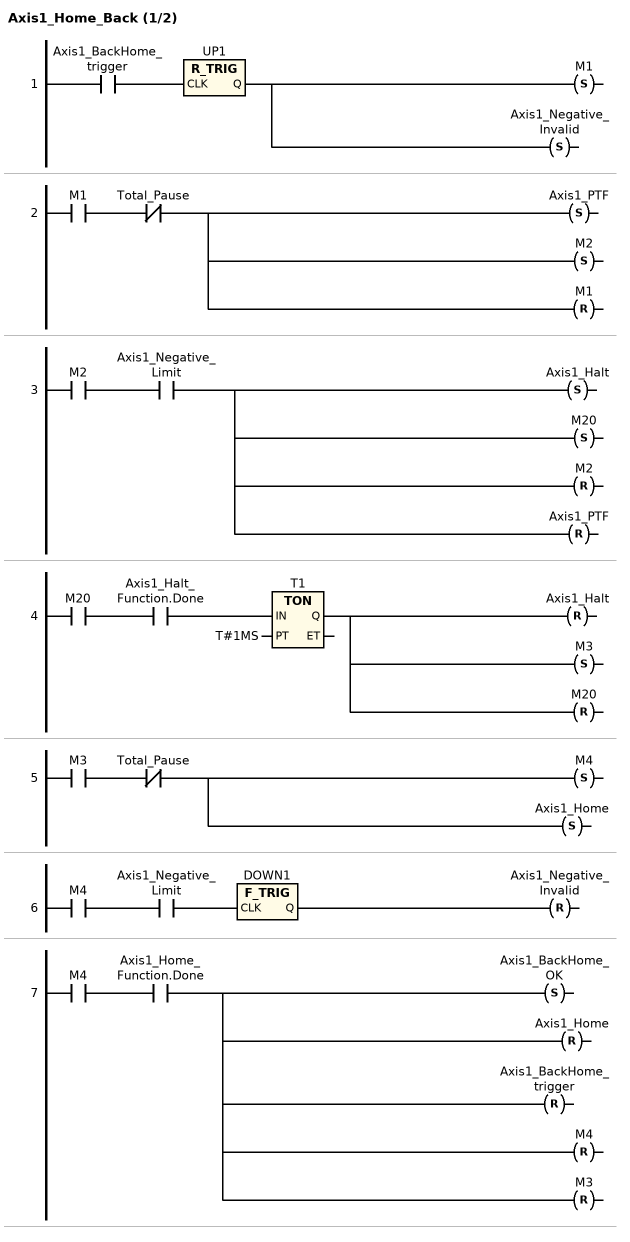
[picture p72: Axis1_Home_Back (LD)]
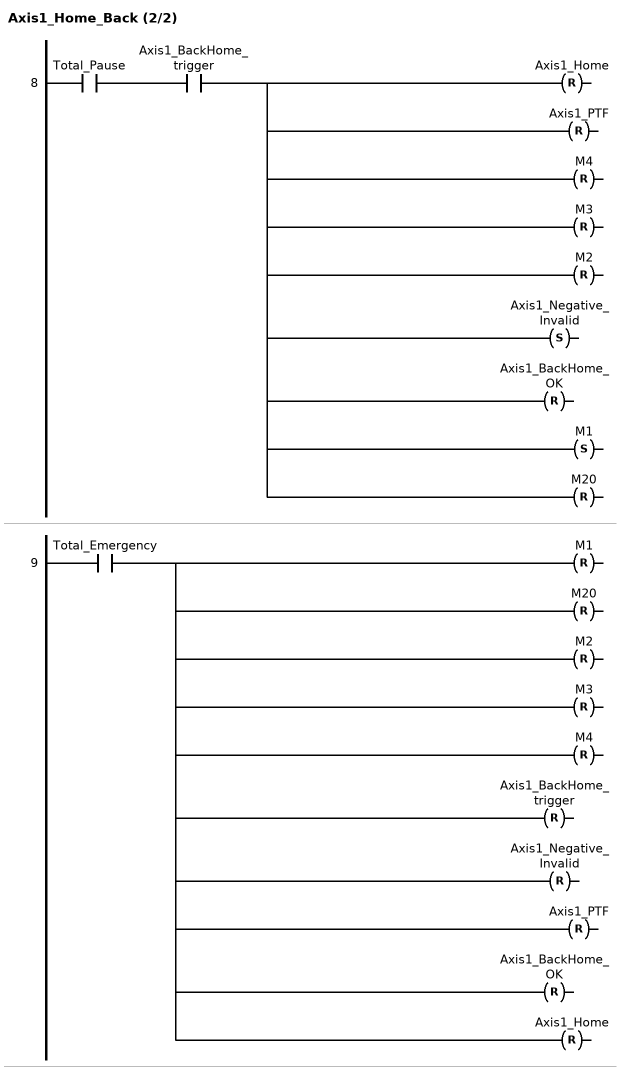
_LD_ (* Ladder Diagram *)
NETWORK 1
	[Axis1_BackHome_trigger] - UP1:R_TRIG(CLK: *) --- (S M1) (S Axis1_Negative_Invalid)
NETWORK 2
	[M1] - [/Total_Pause] --- (S Axis1_PTF) (S M2) (R M1)
NETWORK 3
	[M2] - [Axis1_Negative_Limit] --- (S Axis1_Halt) (S M20) (R M2) (R Axis1_PTF)
NETWORK 4
	[M20] - [Axis1_Halt_Function.Done] - T1:TON(IN: *, PT: T#1MS) --- (R Axis1_Halt) (S M3) (R M20)
NETWORK 5
	[M3] - [/Total_Pause] --- (S M4) (S Axis1_Home)
NETWORK 6
	[M4] - [Axis1_Negative_Limit] - DOWN1:F_TRIG(CLK: *) --- (R Axis1_Negative_Invalid)
NETWORK 7
	[M4] - [Axis1_Home_Function.Done] --- (S Axis1_BackHome_OK) (R Axis1_Home) (R Axis1_BackHome_trigger) (R M4) (R M3)
NETWORK 8
	[Total_Pause] - [Axis1_BackHome_trigger] --- (R Axis1_Home) (R Axis1_PTF) (R M4) (R M3) (R M2) (S Axis1_Negative_Invalid) (R Axis1_BackHome_OK) (S M1) (R M20)
NETWORK 9
	[Total_Emergency] --- (R M1) (R M20) (R M2) (R M3) (R M4) (R Axis1_BackHome_trigger) (R Axis1_Negative_Invalid) (R Axis1_PTF) (R Axis1_BackHome_OK) (R Axis1_Home)
_END_LD_
(* the same logic as Structured Text *)
(* Network 1 *)
UP1(CLK := Axis1_BackHome_trigger);
IF UP1.Q THEN M1 := TRUE; Axis1_Negative_Invalid := TRUE; END_IF;
(* Network 2 *)
_p1 := M1 AND NOT Total_Pause;
IF _p1 THEN Axis1_PTF := TRUE; M2 := TRUE; M1 := FALSE; END_IF;
(* Network 3 *)
_p2 := M2 AND Axis1_Negative_Limit;
IF _p2 THEN Axis1_Halt := TRUE; M20 := TRUE; M2 := FALSE; Axis1_PTF := FALSE; END_IF;
(* Network 4 *)
T1(IN := M20 AND Axis1_Halt_Function.Done, PT := T#1MS);
IF T1.Q THEN Axis1_Halt := FALSE; M3 := TRUE; M20 := FALSE; END_IF;
(* Network 5 *)
IF M3 AND NOT Total_Pause THEN M4 := TRUE; Axis1_Home := TRUE; END_IF;
(* Network 6 *)
DOWN1(CLK := M4 AND Axis1_Negative_Limit);
IF DOWN1.Q THEN Axis1_Negative_Invalid := FALSE; END_IF;
(* Network 7 *)
_p3 := M4 AND Axis1_Home_Function.Done;
IF _p3 THEN Axis1_BackHome_OK := TRUE; Axis1_Home := FALSE; Axis1_BackHome_trigger := FALSE; M4 := FALSE; M3 := FALSE; END_IF;
(* Network 8 *)
IF Total_Pause AND Axis1_BackHome_trigger THEN Axis1_Home := FALSE; Axis1_PTF := FALSE; M4 := FALSE; M3 := FALSE; M2 := FALSE; Axis1_Negative_Invalid := TRUE; Axis1_BackHome_OK := FALSE; M1 := TRUE; M20 := FALSE; END_IF;
(* Network 9 *)
IF Total_Emergency THEN M1 := FALSE; M20 := FALSE; M2 := FALSE; M3 := FALSE; M4 := FALSE; Axis1_BackHome_trigger := FALSE; Axis1_Negative_Invalid := FALSE; Axis1_PTF := FALSE; Axis1_BackHome_OK := FALSE; Axis1_Home := FALSE; END_IF;
END_PROGRAM

(* POU Other_Folder/Home_Back/Axis2_Home_Back, LD *)
PROGRAM Axis2_Home_Back
VAR
	UP1: R_TRIG;
	M1: BOOL;
	M2: BOOL;
	UP2: R_TRIG;
	T1: TON;
	M3: BOOL;
	M4: BOOL;
	DOWN1: F_TRIG;
	M20: BOOL;
END_VAR
VAR (* helpers for the ST form of the networks *)
	_p1 : BOOL;
	_p2 : BOOL;
	_p3 : BOOL;
END_VAR
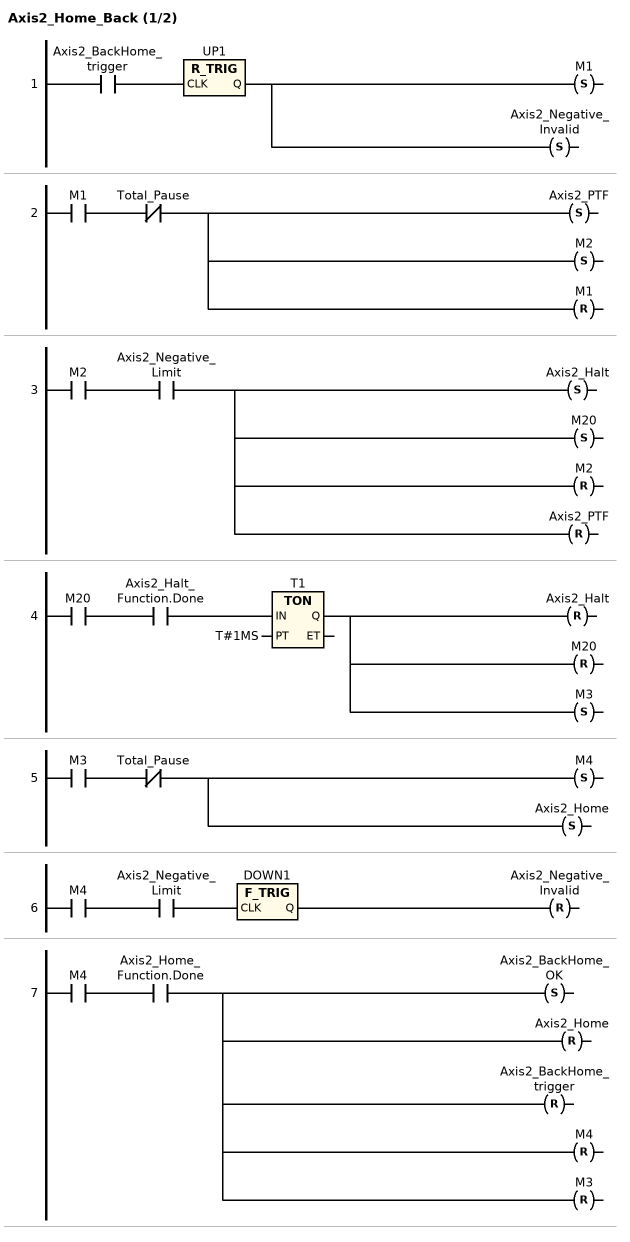
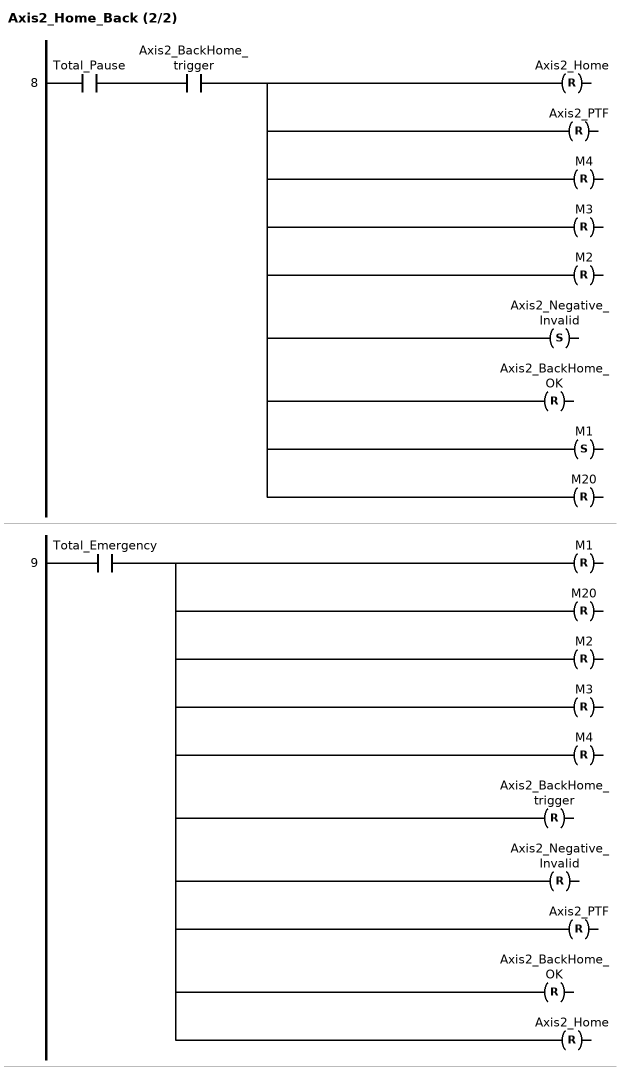
_LD_ (* Ladder Diagram *)
NETWORK 1
	[Axis2_BackHome_trigger] - UP1:R_TRIG(CLK: *) --- (S M1) (S Axis2_Negative_Invalid)
NETWORK 2
	[M1] - [/Total_Pause] --- (S Axis2_PTF) (S M2) (R M1)
NETWORK 3
	[M2] - [Axis2_Negative_Limit] --- (S Axis2_Halt) (S M20) (R M2) (R Axis2_PTF)
NETWORK 4
	[M20] - [Axis2_Halt_Function.Done] - T1:TON(IN: *, PT: T#1MS) --- (R Axis2_Halt) (R M20) (S M3)
NETWORK 5
	[M3] - [/Total_Pause] --- (S M4) (S Axis2_Home)
NETWORK 6
	[M4] - [Axis2_Negative_Limit] - DOWN1:F_TRIG(CLK: *) --- (R Axis2_Negative_Invalid)
NETWORK 7
	[M4] - [Axis2_Home_Function.Done] --- (S Axis2_BackHome_OK) (R Axis2_Home) (R Axis2_BackHome_trigger) (R M4) (R M3)
NETWORK 8
	[Total_Pause] - [Axis2_BackHome_trigger] --- (R Axis2_Home) (R Axis2_PTF) (R M4) (R M3) (R M2) (S Axis2_Negative_Invalid) (R Axis2_BackHome_OK) (S M1) (R M20)
NETWORK 9
	[Total_Emergency] --- (R M1) (R M20) (R M2) (R M3) (R M4) (R Axis2_BackHome_trigger) (R Axis2_Negative_Invalid) (R Axis2_PTF) (R Axis2_BackHome_OK) (R Axis2_Home)
_END_LD_
(* the same logic as Structured Text *)
(* Network 1 *)
UP1(CLK := Axis2_BackHome_trigger);
IF UP1.Q THEN M1 := TRUE; Axis2_Negative_Invalid := TRUE; END_IF;
(* Network 2 *)
_p1 := M1 AND NOT Total_Pause;
IF _p1 THEN Axis2_PTF := TRUE; M2 := TRUE; M1 := FALSE; END_IF;
(* Network 3 *)
_p2 := M2 AND Axis2_Negative_Limit;
IF _p2 THEN Axis2_Halt := TRUE; M20 := TRUE; M2 := FALSE; Axis2_PTF := FALSE; END_IF;
(* Network 4 *)
T1(IN := M20 AND Axis2_Halt_Function.Done, PT := T#1MS);
IF T1.Q THEN Axis2_Halt := FALSE; M20 := FALSE; M3 := TRUE; END_IF;
(* Network 5 *)
IF M3 AND NOT Total_Pause THEN M4 := TRUE; Axis2_Home := TRUE; END_IF;
(* Network 6 *)
DOWN1(CLK := M4 AND Axis2_Negative_Limit);
IF DOWN1.Q THEN Axis2_Negative_Invalid := FALSE; END_IF;
(* Network 7 *)
_p3 := M4 AND Axis2_Home_Function.Done;
IF _p3 THEN Axis2_BackHome_OK := TRUE; Axis2_Home := FALSE; Axis2_BackHome_trigger := FALSE; M4 := FALSE; M3 := FALSE; END_IF;
(* Network 8 *)
IF Total_Pause AND Axis2_BackHome_trigger THEN Axis2_Home := FALSE; Axis2_PTF := FALSE; M4 := FALSE; M3 := FALSE; M2 := FALSE; Axis2_Negative_Invalid := TRUE; Axis2_BackHome_OK := FALSE; M1 := TRUE; M20 := FALSE; END_IF;
(* Network 9 *)
IF Total_Emergency THEN M1 := FALSE; M20 := FALSE; M2 := FALSE; M3 := FALSE; M4 := FALSE; Axis2_BackHome_trigger := FALSE; Axis2_Negative_Invalid := FALSE; Axis2_PTF := FALSE; Axis2_BackHome_OK := FALSE; Axis2_Home := FALSE; END_IF;
END_PROGRAM

(* POU Other_Folder/Home_Back/Axis3_Home_Back, LD *)
PROGRAM Axis3_Home_Back
VAR
	UP1: R_TRIG;
	M1: BOOL;
	M2: BOOL;
	UP2: R_TRIG;
	T1: TON;
	M3: BOOL;
	M4: BOOL;
	DOWN1: F_TRIG;
	M20: BOOL;
END_VAR
VAR (* helpers for the ST form of the networks *)
	_p1 : BOOL;
	_p2 : BOOL;
	_p3 : BOOL;
END_VAR
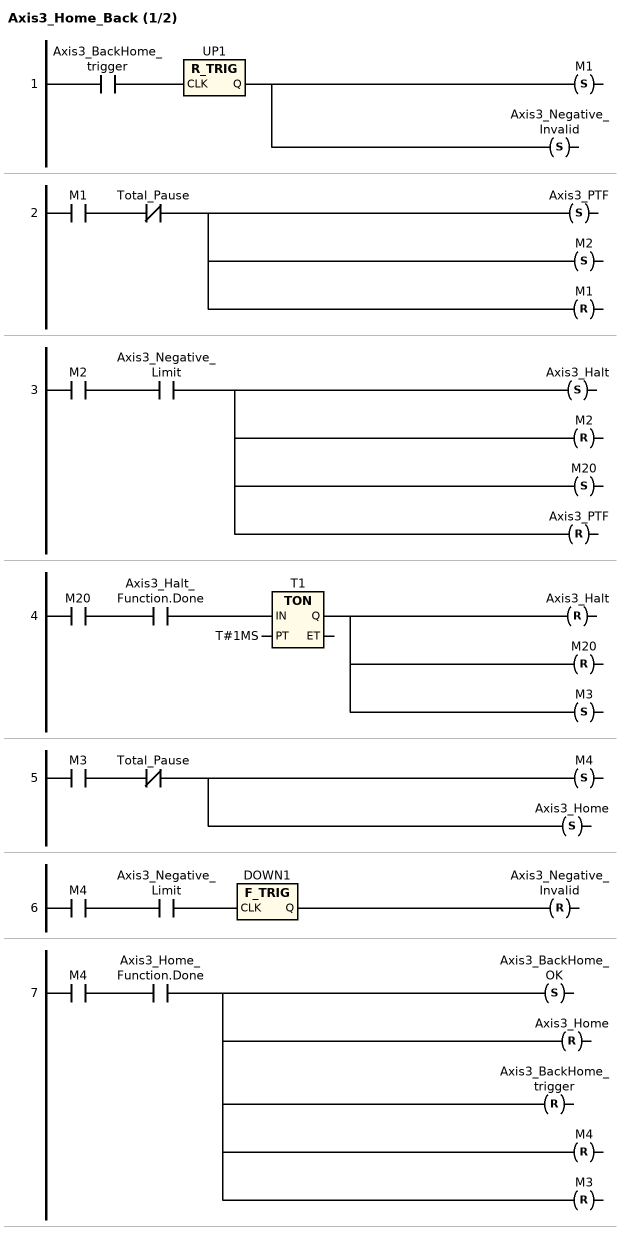
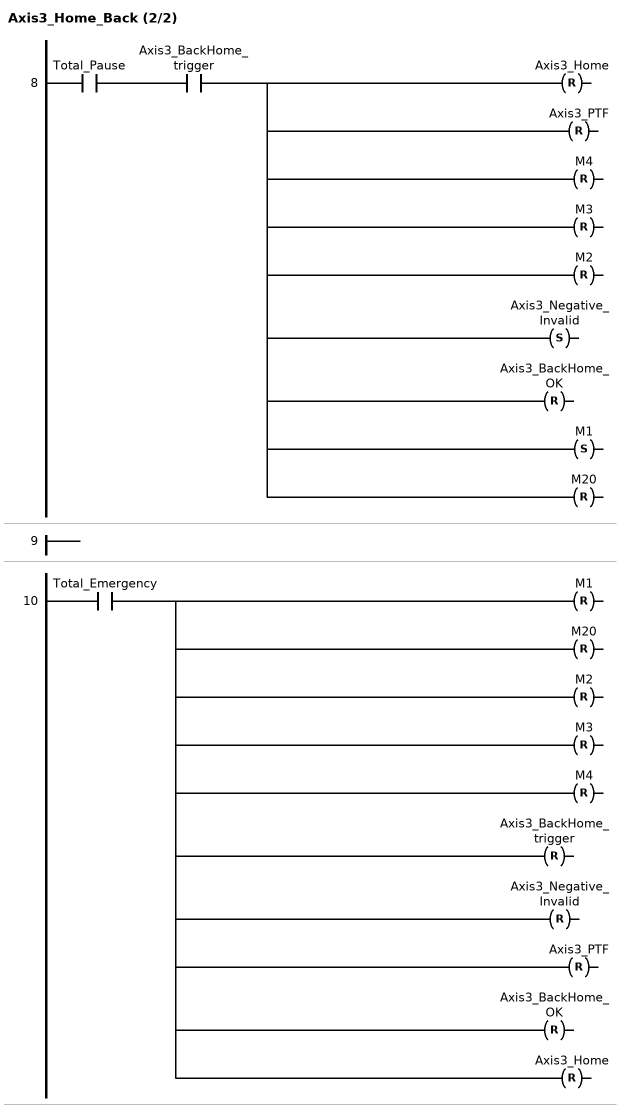
_LD_ (* Ladder Diagram *)
NETWORK 1
	[Axis3_BackHome_trigger] - UP1:R_TRIG(CLK: *) --- (S M1) (S Axis3_Negative_Invalid)
NETWORK 2
	[M1] - [/Total_Pause] --- (S Axis3_PTF) (S M2) (R M1)
NETWORK 3
	[M2] - [Axis3_Negative_Limit] --- (S Axis3_Halt) (R M2) (S M20) (R Axis3_PTF)
NETWORK 4
	[M20] - [Axis3_Halt_Function.Done] - T1:TON(IN: *, PT: T#1MS) --- (R Axis3_Halt) (R M20) (S M3)
NETWORK 5
	[M3] - [/Total_Pause] --- (S M4) (S Axis3_Home)
NETWORK 6
	[M4] - [Axis3_Negative_Limit] - DOWN1:F_TRIG(CLK: *) --- (R Axis3_Negative_Invalid)
NETWORK 7
	[M4] - [Axis3_Home_Function.Done] --- (S Axis3_BackHome_OK) (R Axis3_Home) (R Axis3_BackHome_trigger) (R M4) (R M3)
NETWORK 8
	[Total_Pause] - [Axis3_BackHome_trigger] --- (R Axis3_Home) (R Axis3_PTF) (R M4) (R M3) (R M2) (S Axis3_Negative_Invalid) (R Axis3_BackHome_OK) (S M1) (R M20)
NETWORK 9
	*
NETWORK 10
	[Total_Emergency] --- (R M1) (R M20) (R M2) (R M3) (R M4) (R Axis3_BackHome_trigger) (R Axis3_Negative_Invalid) (R Axis3_PTF) (R Axis3_BackHome_OK) (R Axis3_Home)
_END_LD_
(* the same logic as Structured Text *)
(* Network 1 *)
UP1(CLK := Axis3_BackHome_trigger);
IF UP1.Q THEN M1 := TRUE; Axis3_Negative_Invalid := TRUE; END_IF;
(* Network 2 *)
_p1 := M1 AND NOT Total_Pause;
IF _p1 THEN Axis3_PTF := TRUE; M2 := TRUE; M1 := FALSE; END_IF;
(* Network 3 *)
_p2 := M2 AND Axis3_Negative_Limit;
IF _p2 THEN Axis3_Halt := TRUE; M2 := FALSE; M20 := TRUE; Axis3_PTF := FALSE; END_IF;
(* Network 4 *)
T1(IN := M20 AND Axis3_Halt_Function.Done, PT := T#1MS);
IF T1.Q THEN Axis3_Halt := FALSE; M20 := FALSE; M3 := TRUE; END_IF;
(* Network 5 *)
IF M3 AND NOT Total_Pause THEN M4 := TRUE; Axis3_Home := TRUE; END_IF;
(* Network 6 *)
DOWN1(CLK := M4 AND Axis3_Negative_Limit);
IF DOWN1.Q THEN Axis3_Negative_Invalid := FALSE; END_IF;
(* Network 7 *)
_p3 := M4 AND Axis3_Home_Function.Done;
IF _p3 THEN Axis3_BackHome_OK := TRUE; Axis3_Home := FALSE; Axis3_BackHome_trigger := FALSE; M4 := FALSE; M3 := FALSE; END_IF;
(* Network 8 *)
IF Total_Pause AND Axis3_BackHome_trigger THEN Axis3_Home := FALSE; Axis3_PTF := FALSE; M4 := FALSE; M3 := FALSE; M2 := FALSE; Axis3_Negative_Invalid := TRUE; Axis3_BackHome_OK := FALSE; M1 := TRUE; M20 := FALSE; END_IF;
(* Network 9 *)
(* Network 10 *)
IF Total_Emergency THEN M1 := FALSE; M20 := FALSE; M2 := FALSE; M3 := FALSE; M4 := FALSE; Axis3_BackHome_trigger := FALSE; Axis3_Negative_Invalid := FALSE; Axis3_PTF := FALSE; Axis3_BackHome_OK := FALSE; Axis3_Home := FALSE; END_IF;
END_PROGRAM

(* POU Other_Folder/Home_Back/Axis4_Home_Back, LD *)
PROGRAM Axis4_Home_Back
VAR
	UP1: R_TRIG;
	M1: BOOL;
	M2: BOOL;
	UP2: R_TRIG;
	T1: TON;
	M3: BOOL;
	M4: BOOL;
	DOWN1: F_TRIG;
	M20: BOOL;
END_VAR
VAR (* helpers for the ST form of the networks *)
	_p1 : BOOL;
	_p2 : BOOL;
	_p3 : BOOL;
END_VAR
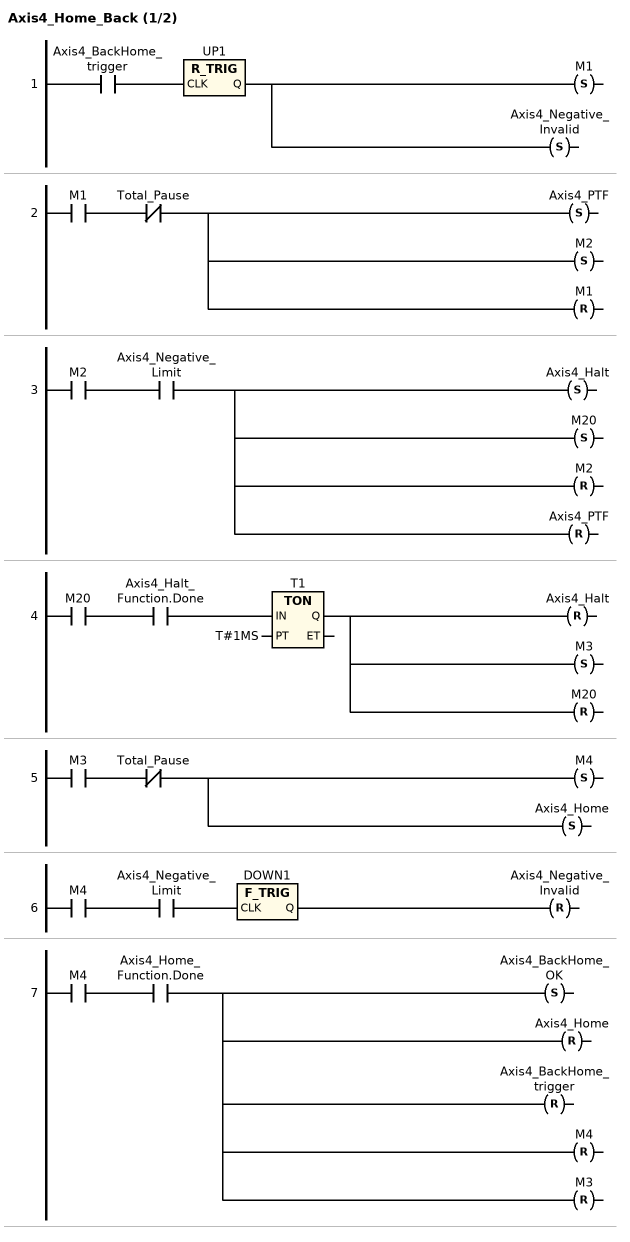
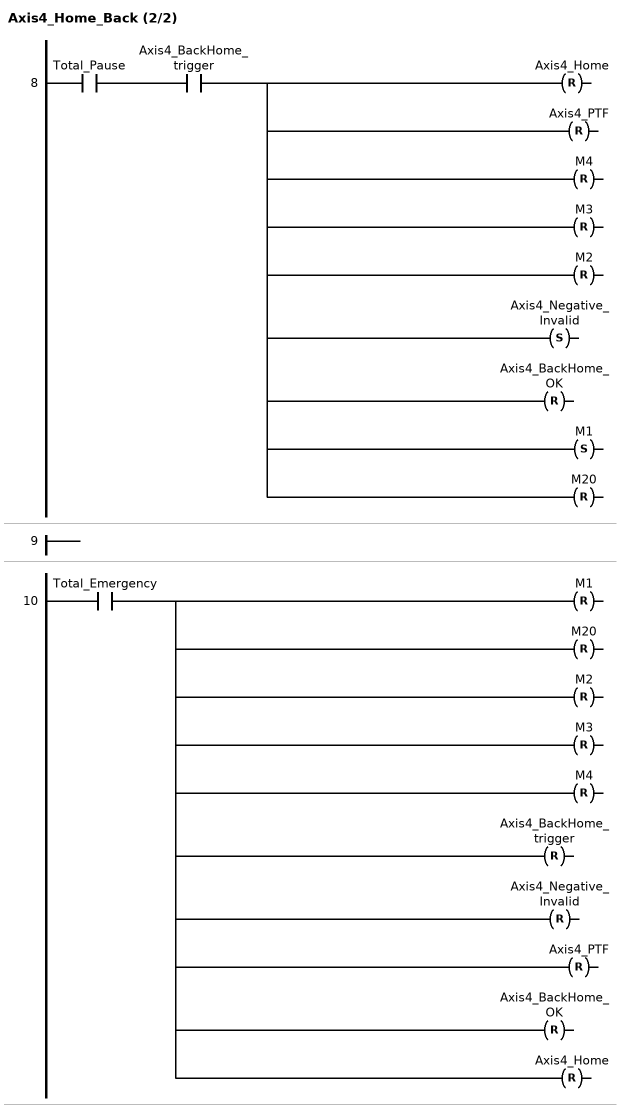
_LD_ (* Ladder Diagram *)
NETWORK 1
	[Axis4_BackHome_trigger] - UP1:R_TRIG(CLK: *) --- (S M1) (S Axis4_Negative_Invalid)
NETWORK 2
	[M1] - [/Total_Pause] --- (S Axis4_PTF) (S M2) (R M1)
NETWORK 3
	[M2] - [Axis4_Negative_Limit] --- (S Axis4_Halt) (S M20) (R M2) (R Axis4_PTF)
NETWORK 4
	[M20] - [Axis4_Halt_Function.Done] - T1:TON(IN: *, PT: T#1MS) --- (R Axis4_Halt) (S M3) (R M20)
NETWORK 5
	[M3] - [/Total_Pause] --- (S M4) (S Axis4_Home)
NETWORK 6
	[M4] - [Axis4_Negative_Limit] - DOWN1:F_TRIG(CLK: *) --- (R Axis4_Negative_Invalid)
NETWORK 7
	[M4] - [Axis4_Home_Function.Done] --- (S Axis4_BackHome_OK) (R Axis4_Home) (R Axis4_BackHome_trigger) (R M4) (R M3)
NETWORK 8
	[Total_Pause] - [Axis4_BackHome_trigger] --- (R Axis4_Home) (R Axis4_PTF) (R M4) (R M3) (R M2) (S Axis4_Negative_Invalid) (R Axis4_BackHome_OK) (S M1) (R M20)
NETWORK 9
	*
NETWORK 10
	[Total_Emergency] --- (R M1) (R M20) (R M2) (R M3) (R M4) (R Axis4_BackHome_trigger) (R Axis4_Negative_Invalid) (R Axis4_PTF) (R Axis4_BackHome_OK) (R Axis4_Home)
_END_LD_
(* the same logic as Structured Text *)
(* Network 1 *)
UP1(CLK := Axis4_BackHome_trigger);
IF UP1.Q THEN M1 := TRUE; Axis4_Negative_Invalid := TRUE; END_IF;
(* Network 2 *)
_p1 := M1 AND NOT Total_Pause;
IF _p1 THEN Axis4_PTF := TRUE; M2 := TRUE; M1 := FALSE; END_IF;
(* Network 3 *)
_p2 := M2 AND Axis4_Negative_Limit;
IF _p2 THEN Axis4_Halt := TRUE; M20 := TRUE; M2 := FALSE; Axis4_PTF := FALSE; END_IF;
(* Network 4 *)
T1(IN := M20 AND Axis4_Halt_Function.Done, PT := T#1MS);
IF T1.Q THEN Axis4_Halt := FALSE; M3 := TRUE; M20 := FALSE; END_IF;
(* Network 5 *)
IF M3 AND NOT Total_Pause THEN M4 := TRUE; Axis4_Home := TRUE; END_IF;
(* Network 6 *)
DOWN1(CLK := M4 AND Axis4_Negative_Limit);
IF DOWN1.Q THEN Axis4_Negative_Invalid := FALSE; END_IF;
(* Network 7 *)
_p3 := M4 AND Axis4_Home_Function.Done;
IF _p3 THEN Axis4_BackHome_OK := TRUE; Axis4_Home := FALSE; Axis4_BackHome_trigger := FALSE; M4 := FALSE; M3 := FALSE; END_IF;
(* Network 8 *)
IF Total_Pause AND Axis4_BackHome_trigger THEN Axis4_Home := FALSE; Axis4_PTF := FALSE; M4 := FALSE; M3 := FALSE; M2 := FALSE; Axis4_Negative_Invalid := TRUE; Axis4_BackHome_OK := FALSE; M1 := TRUE; M20 := FALSE; END_IF;
(* Network 9 *)
(* Network 10 *)
IF Total_Emergency THEN M1 := FALSE; M20 := FALSE; M2 := FALSE; M3 := FALSE; M4 := FALSE; Axis4_BackHome_trigger := FALSE; Axis4_Negative_Invalid := FALSE; Axis4_PTF := FALSE; Axis4_BackHome_OK := FALSE; Axis4_Home := FALSE; END_IF;
END_PROGRAM

(* POU Other_Folder/Home_Back/Axis5_Home_Back, LD *)
PROGRAM Axis5_Home_Back
VAR
	UP1: R_TRIG;
	M1: BOOL;
	M2: BOOL;
	UP2: R_TRIG;
	T1: TON;
	M3: BOOL;
	M4: BOOL;
	DOWN1: F_TRIG;
	M20: BOOL;
END_VAR
VAR (* helpers for the ST form of the networks *)
	_p1 : BOOL;
	_p2 : BOOL;
	_p3 : BOOL;
END_VAR
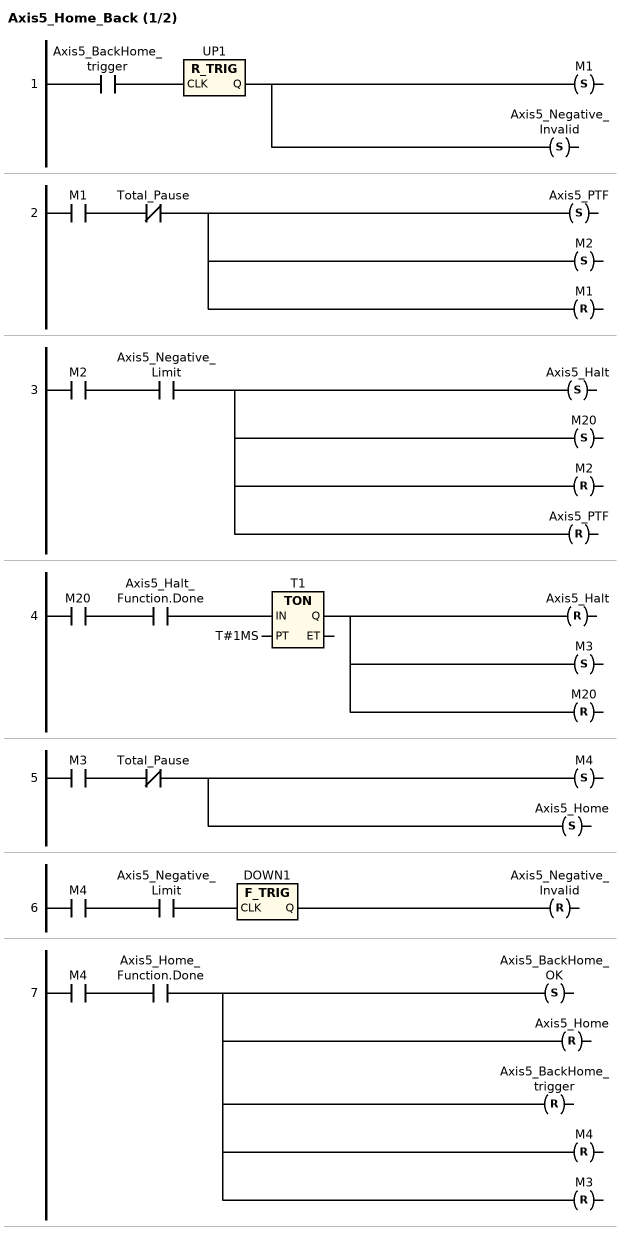
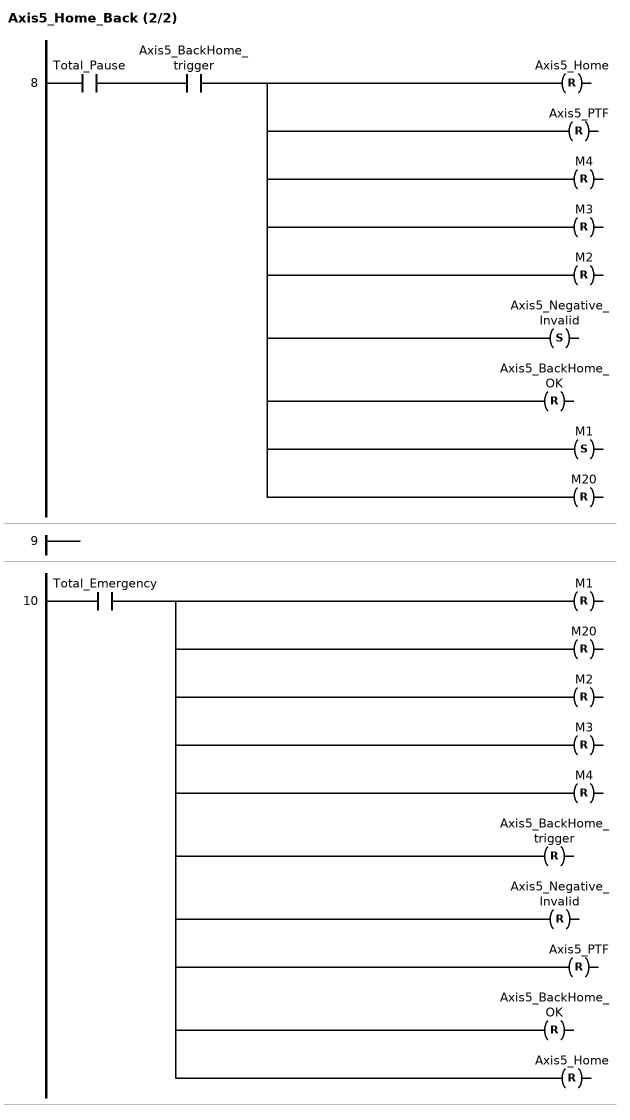
_LD_ (* Ladder Diagram *)
NETWORK 1
	[Axis5_BackHome_trigger] - UP1:R_TRIG(CLK: *) --- (S M1) (S Axis5_Negative_Invalid)
NETWORK 2
	[M1] - [/Total_Pause] --- (S Axis5_PTF) (S M2) (R M1)
NETWORK 3
	[M2] - [Axis5_Negative_Limit] --- (S Axis5_Halt) (S M20) (R M2) (R Axis5_PTF)
NETWORK 4
	[M20] - [Axis5_Halt_Function.Done] - T1:TON(IN: *, PT: T#1MS) --- (R Axis5_Halt) (S M3) (R M20)
NETWORK 5
	[M3] - [/Total_Pause] --- (S M4) (S Axis5_Home)
NETWORK 6
	[M4] - [Axis5_Negative_Limit] - DOWN1:F_TRIG(CLK: *) --- (R Axis5_Negative_Invalid)
NETWORK 7
	[M4] - [Axis5_Home_Function.Done] --- (S Axis5_BackHome_OK) (R Axis5_Home) (R Axis5_BackHome_trigger) (R M4) (R M3)
NETWORK 8
	[Total_Pause] - [Axis5_BackHome_trigger] --- (R Axis5_Home) (R Axis5_PTF) (R M4) (R M3) (R M2) (S Axis5_Negative_Invalid) (R Axis5_BackHome_OK) (S M1) (R M20)
NETWORK 9
	*
NETWORK 10
	[Total_Emergency] --- (R M1) (R M20) (R M2) (R M3) (R M4) (R Axis5_BackHome_trigger) (R Axis5_Negative_Invalid) (R Axis5_PTF) (R Axis5_BackHome_OK) (R Axis5_Home)
_END_LD_
(* the same logic as Structured Text *)
(* Network 1 *)
UP1(CLK := Axis5_BackHome_trigger);
IF UP1.Q THEN M1 := TRUE; Axis5_Negative_Invalid := TRUE; END_IF;
(* Network 2 *)
_p1 := M1 AND NOT Total_Pause;
IF _p1 THEN Axis5_PTF := TRUE; M2 := TRUE; M1 := FALSE; END_IF;
(* Network 3 *)
_p2 := M2 AND Axis5_Negative_Limit;
IF _p2 THEN Axis5_Halt := TRUE; M20 := TRUE; M2 := FALSE; Axis5_PTF := FALSE; END_IF;
(* Network 4 *)
T1(IN := M20 AND Axis5_Halt_Function.Done, PT := T#1MS);
IF T1.Q THEN Axis5_Halt := FALSE; M3 := TRUE; M20 := FALSE; END_IF;
(* Network 5 *)
IF M3 AND NOT Total_Pause THEN M4 := TRUE; Axis5_Home := TRUE; END_IF;
(* Network 6 *)
DOWN1(CLK := M4 AND Axis5_Negative_Limit);
IF DOWN1.Q THEN Axis5_Negative_Invalid := FALSE; END_IF;
(* Network 7 *)
_p3 := M4 AND Axis5_Home_Function.Done;
IF _p3 THEN Axis5_BackHome_OK := TRUE; Axis5_Home := FALSE; Axis5_BackHome_trigger := FALSE; M4 := FALSE; M3 := FALSE; END_IF;
(* Network 8 *)
IF Total_Pause AND Axis5_BackHome_trigger THEN Axis5_Home := FALSE; Axis5_PTF := FALSE; M4 := FALSE; M3 := FALSE; M2 := FALSE; Axis5_Negative_Invalid := TRUE; Axis5_BackHome_OK := FALSE; M1 := TRUE; M20 := FALSE; END_IF;
(* Network 9 *)
(* Network 10 *)
IF Total_Emergency THEN M1 := FALSE; M20 := FALSE; M2 := FALSE; M3 := FALSE; M4 := FALSE; Axis5_BackHome_trigger := FALSE; Axis5_Negative_Invalid := FALSE; Axis5_PTF := FALSE; Axis5_BackHome_OK := FALSE; Axis5_Home := FALSE; END_IF;
END_PROGRAM

(* POU Other_Folder/Home_Back/Axis6_Home_Back, LD *)
PROGRAM Axis6_Home_Back
VAR
	UP1: R_TRIG;
	M1: BOOL;
	M2: BOOL;
	UP2: R_TRIG;
	T1: TON;
	M3: BOOL;
	M4: BOOL;
	DOWN1: F_TRIG;
	M20: BOOL;
END_VAR
VAR (* helpers for the ST form of the networks *)
	_p1 : BOOL;
	_p2 : BOOL;
	_p3 : BOOL;
END_VAR
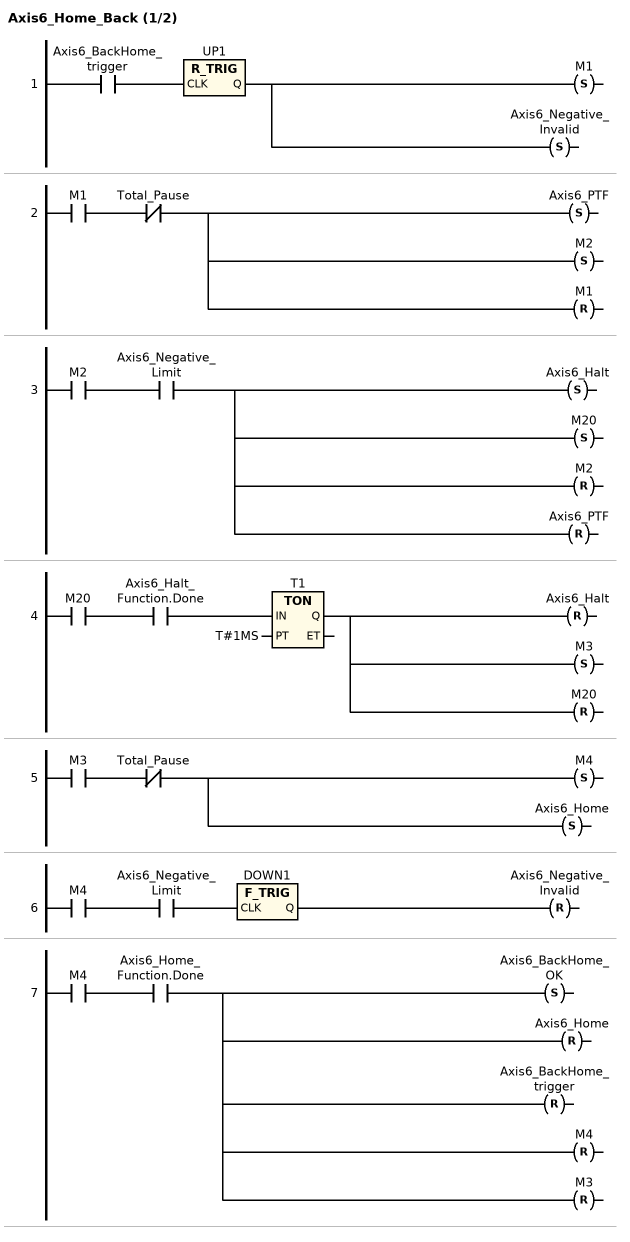
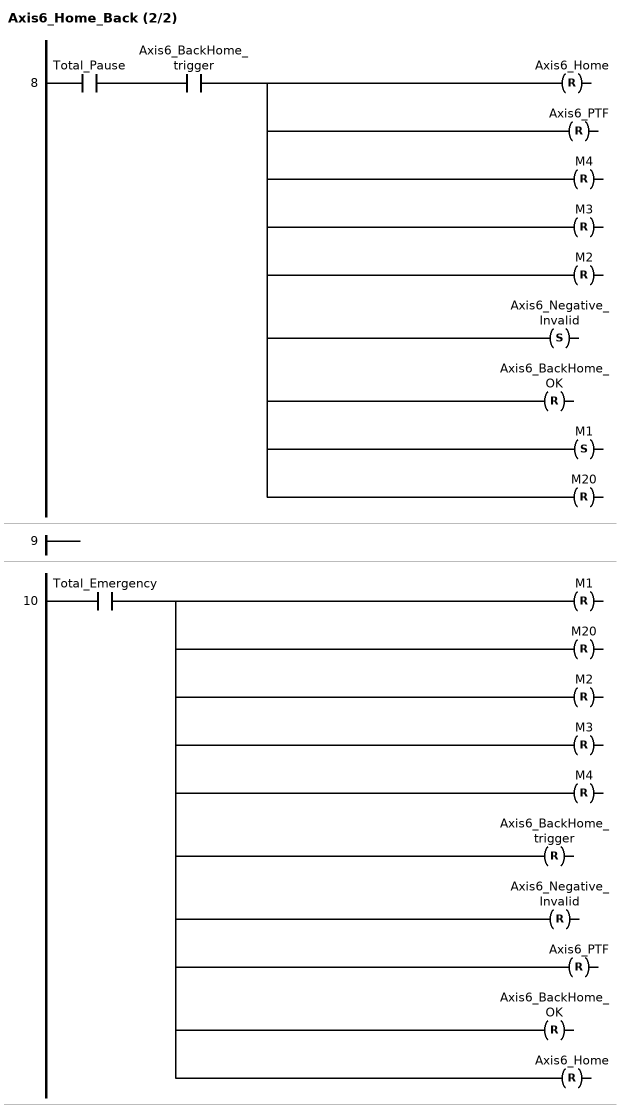
_LD_ (* Ladder Diagram *)
NETWORK 1
	[Axis6_BackHome_trigger] - UP1:R_TRIG(CLK: *) --- (S M1) (S Axis6_Negative_Invalid)
NETWORK 2
	[M1] - [/Total_Pause] --- (S Axis6_PTF) (S M2) (R M1)
NETWORK 3
	[M2] - [Axis6_Negative_Limit] --- (S Axis6_Halt) (S M20) (R M2) (R Axis6_PTF)
NETWORK 4
	[M20] - [Axis6_Halt_Function.Done] - T1:TON(IN: *, PT: T#1MS) --- (R Axis6_Halt) (S M3) (R M20)
NETWORK 5
	[M3] - [/Total_Pause] --- (S M4) (S Axis6_Home)
NETWORK 6
	[M4] - [Axis6_Negative_Limit] - DOWN1:F_TRIG(CLK: *) --- (R Axis6_Negative_Invalid)
NETWORK 7
	[M4] - [Axis6_Home_Function.Done] --- (S Axis6_BackHome_OK) (R Axis6_Home) (R Axis6_BackHome_trigger) (R M4) (R M3)
NETWORK 8
	[Total_Pause] - [Axis6_BackHome_trigger] --- (R Axis6_Home) (R Axis6_PTF) (R M4) (R M3) (R M2) (S Axis6_Negative_Invalid) (R Axis6_BackHome_OK) (S M1) (R M20)
NETWORK 9
	*
NETWORK 10
	[Total_Emergency] --- (R M1) (R M20) (R M2) (R M3) (R M4) (R Axis6_BackHome_trigger) (R Axis6_Negative_Invalid) (R Axis6_PTF) (R Axis6_BackHome_OK) (R Axis6_Home)
_END_LD_
(* the same logic as Structured Text *)
(* Network 1 *)
UP1(CLK := Axis6_BackHome_trigger);
IF UP1.Q THEN M1 := TRUE; Axis6_Negative_Invalid := TRUE; END_IF;
(* Network 2 *)
_p1 := M1 AND NOT Total_Pause;
IF _p1 THEN Axis6_PTF := TRUE; M2 := TRUE; M1 := FALSE; END_IF;
(* Network 3 *)
_p2 := M2 AND Axis6_Negative_Limit;
IF _p2 THEN Axis6_Halt := TRUE; M20 := TRUE; M2 := FALSE; Axis6_PTF := FALSE; END_IF;
(* Network 4 *)
T1(IN := M20 AND Axis6_Halt_Function.Done, PT := T#1MS);
IF T1.Q THEN Axis6_Halt := FALSE; M3 := TRUE; M20 := FALSE; END_IF;
(* Network 5 *)
IF M3 AND NOT Total_Pause THEN M4 := TRUE; Axis6_Home := TRUE; END_IF;
(* Network 6 *)
DOWN1(CLK := M4 AND Axis6_Negative_Limit);
IF DOWN1.Q THEN Axis6_Negative_Invalid := FALSE; END_IF;
(* Network 7 *)
_p3 := M4 AND Axis6_Home_Function.Done;
IF _p3 THEN Axis6_BackHome_OK := TRUE; Axis6_Home := FALSE; Axis6_BackHome_trigger := FALSE; M4 := FALSE; M3 := FALSE; END_IF;
(* Network 8 *)
IF Total_Pause AND Axis6_BackHome_trigger THEN Axis6_Home := FALSE; Axis6_PTF := FALSE; M4 := FALSE; M3 := FALSE; M2 := FALSE; Axis6_Negative_Invalid := TRUE; Axis6_BackHome_OK := FALSE; M1 := TRUE; M20 := FALSE; END_IF;
(* Network 9 *)
(* Network 10 *)
IF Total_Emergency THEN M1 := FALSE; M20 := FALSE; M2 := FALSE; M3 := FALSE; M4 := FALSE; Axis6_BackHome_trigger := FALSE; Axis6_Negative_Invalid := FALSE; Axis6_PTF := FALSE; Axis6_BackHome_OK := FALSE; Axis6_Home := FALSE; END_IF;
END_PROGRAM

(* POU Other_Folder/Home_Back/Axis7_Home_Back, LD *)
PROGRAM Axis7_Home_Back
VAR
	UP1: R_TRIG;
	M1: BOOL;
	M2: BOOL;
	UP2: R_TRIG;
	T1: TON;
	M3: BOOL;
	M4: BOOL;
	DOWN1: F_TRIG;
	M20: BOOL;
END_VAR
VAR (* helpers for the ST form of the networks *)
	_p1 : BOOL;
	_p2 : BOOL;
	_p3 : BOOL;
END_VAR
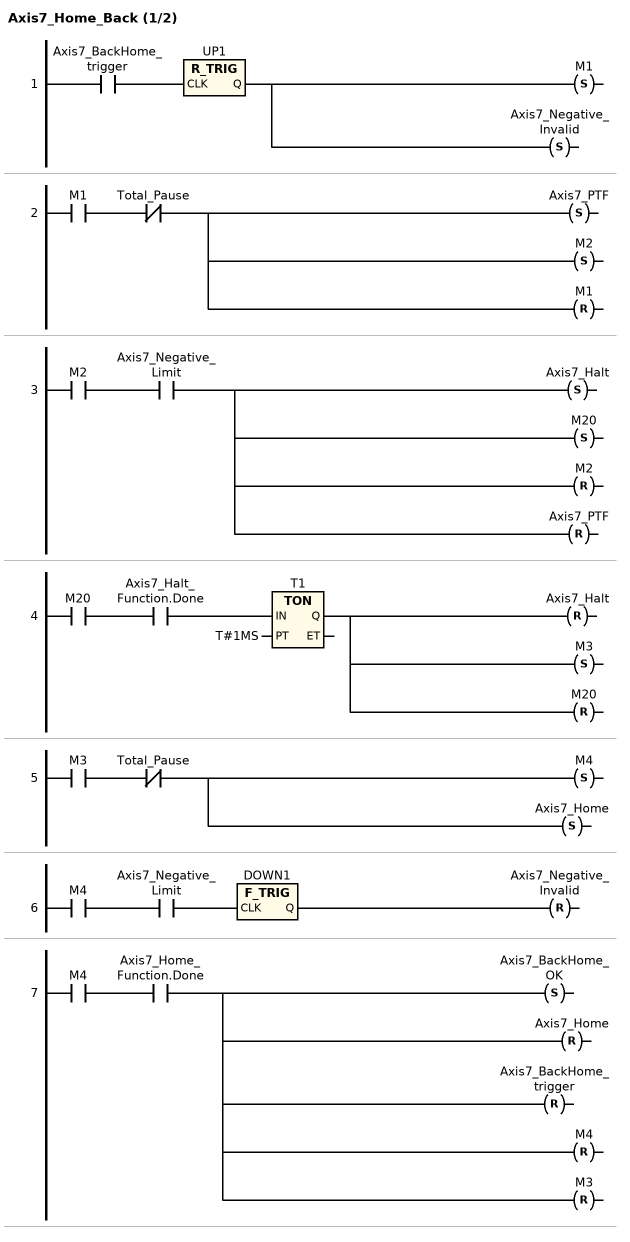
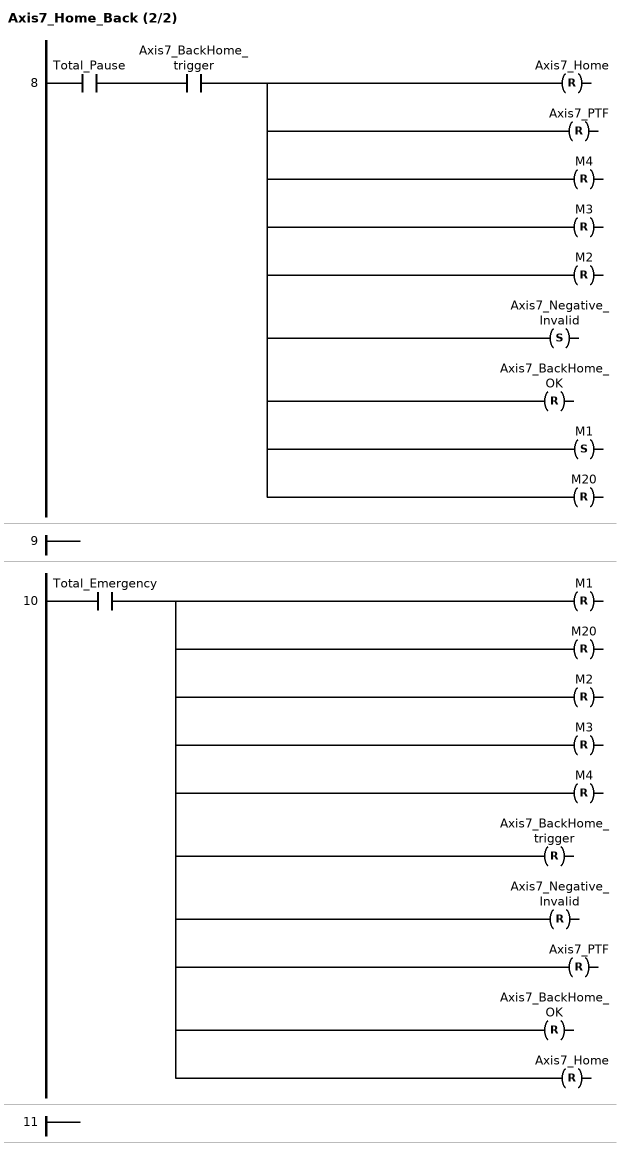
_LD_ (* Ladder Diagram *)
NETWORK 1
	[Axis7_BackHome_trigger] - UP1:R_TRIG(CLK: *) --- (S M1) (S Axis7_Negative_Invalid)
NETWORK 2
	[M1] - [/Total_Pause] --- (S Axis7_PTF) (S M2) (R M1)
NETWORK 3
	[M2] - [Axis7_Negative_Limit] --- (S Axis7_Halt) (S M20) (R M2) (R Axis7_PTF)
NETWORK 4
	[M20] - [Axis7_Halt_Function.Done] - T1:TON(IN: *, PT: T#1MS) --- (R Axis7_Halt) (S M3) (R M20)
NETWORK 5
	[M3] - [/Total_Pause] --- (S M4) (S Axis7_Home)
NETWORK 6
	[M4] - [Axis7_Negative_Limit] - DOWN1:F_TRIG(CLK: *) --- (R Axis7_Negative_Invalid)
NETWORK 7
	[M4] - [Axis7_Home_Function.Done] --- (S Axis7_BackHome_OK) (R Axis7_Home) (R Axis7_BackHome_trigger) (R M4) (R M3)
NETWORK 8
	[Total_Pause] - [Axis7_BackHome_trigger] --- (R Axis7_Home) (R Axis7_PTF) (R M4) (R M3) (R M2) (S Axis7_Negative_Invalid) (R Axis7_BackHome_OK) (S M1) (R M20)
NETWORK 9
	*
NETWORK 10
	[Total_Emergency] --- (R M1) (R M20) (R M2) (R M3) (R M4) (R Axis7_BackHome_trigger) (R Axis7_Negative_Invalid) (R Axis7_PTF) (R Axis7_BackHome_OK) (R Axis7_Home)
NETWORK 11
	*
_END_LD_
(* the same logic as Structured Text *)
(* Network 1 *)
UP1(CLK := Axis7_BackHome_trigger);
IF UP1.Q THEN M1 := TRUE; Axis7_Negative_Invalid := TRUE; END_IF;
(* Network 2 *)
_p1 := M1 AND NOT Total_Pause;
IF _p1 THEN Axis7_PTF := TRUE; M2 := TRUE; M1 := FALSE; END_IF;
(* Network 3 *)
_p2 := M2 AND Axis7_Negative_Limit;
IF _p2 THEN Axis7_Halt := TRUE; M20 := TRUE; M2 := FALSE; Axis7_PTF := FALSE; END_IF;
(* Network 4 *)
T1(IN := M20 AND Axis7_Halt_Function.Done, PT := T#1MS);
IF T1.Q THEN Axis7_Halt := FALSE; M3 := TRUE; M20 := FALSE; END_IF;
(* Network 5 *)
IF M3 AND NOT Total_Pause THEN M4 := TRUE; Axis7_Home := TRUE; END_IF;
(* Network 6 *)
DOWN1(CLK := M4 AND Axis7_Negative_Limit);
IF DOWN1.Q THEN Axis7_Negative_Invalid := FALSE; END_IF;
(* Network 7 *)
_p3 := M4 AND Axis7_Home_Function.Done;
IF _p3 THEN Axis7_BackHome_OK := TRUE; Axis7_Home := FALSE; Axis7_BackHome_trigger := FALSE; M4 := FALSE; M3 := FALSE; END_IF;
(* Network 8 *)
IF Total_Pause AND Axis7_BackHome_trigger THEN Axis7_Home := FALSE; Axis7_PTF := FALSE; M4 := FALSE; M3 := FALSE; M2 := FALSE; Axis7_Negative_Invalid := TRUE; Axis7_BackHome_OK := FALSE; M1 := TRUE; M20 := FALSE; END_IF;
(* Network 9 *)
(* Network 10 *)
IF Total_Emergency THEN M1 := FALSE; M20 := FALSE; M2 := FALSE; M3 := FALSE; M4 := FALSE; Axis7_BackHome_trigger := FALSE; Axis7_Negative_Invalid := FALSE; Axis7_PTF := FALSE; Axis7_BackHome_OK := FALSE; Axis7_Home := FALSE; END_IF;
(* Network 11 *)
END_PROGRAM

(* POU Other_Folder/Home_Back/Axis8_Home_Back, LD *)
PROGRAM Axis8_Home_Back
VAR
	UP1: R_TRIG;
	M1: BOOL;
	M2: BOOL;
	UP2: R_TRIG;
	T1: TON;
	M3: BOOL;
	M4: BOOL;
	DOWN1: F_TRIG;
	M20: BOOL;
END_VAR
VAR (* helpers for the ST form of the networks *)
	_p1 : BOOL;
	_p2 : BOOL;
	_p3 : BOOL;
END_VAR
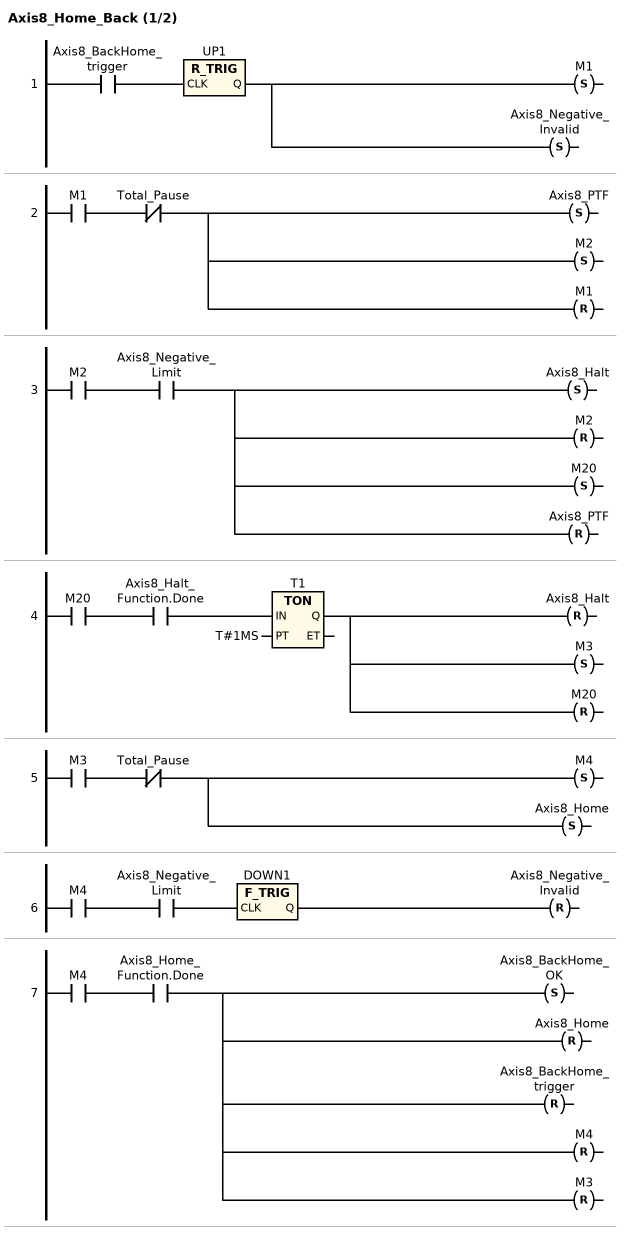
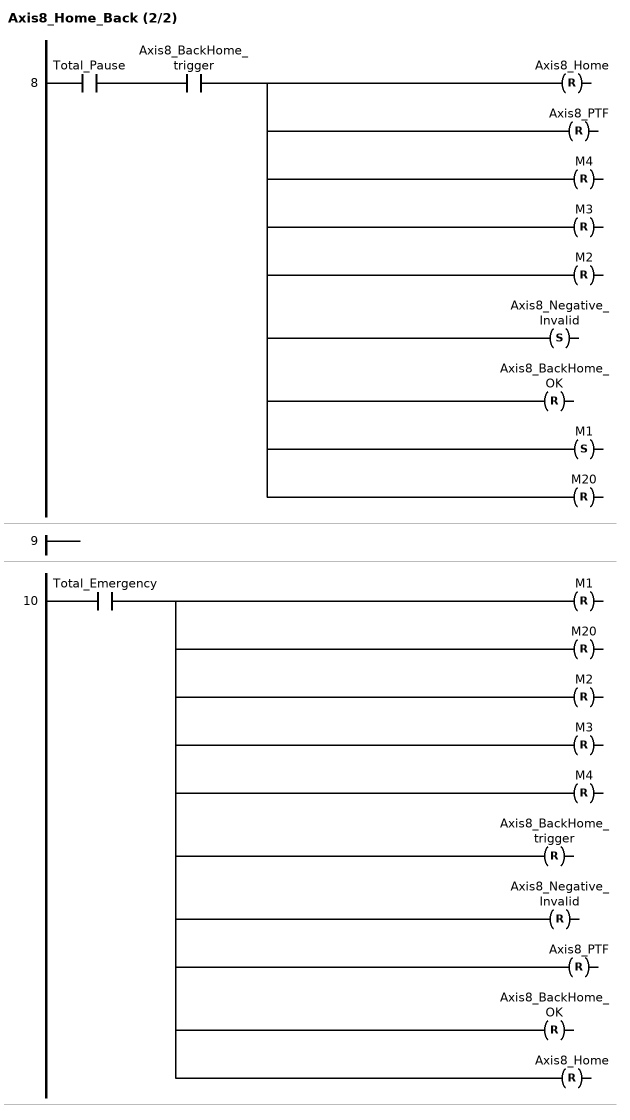
_LD_ (* Ladder Diagram *)
NETWORK 1
	[Axis8_BackHome_trigger] - UP1:R_TRIG(CLK: *) --- (S M1) (S Axis8_Negative_Invalid)
NETWORK 2
	[M1] - [/Total_Pause] --- (S Axis8_PTF) (S M2) (R M1)
NETWORK 3
	[M2] - [Axis8_Negative_Limit] --- (S Axis8_Halt) (R M2) (S M20) (R Axis8_PTF)
NETWORK 4
	[M20] - [Axis8_Halt_Function.Done] - T1:TON(IN: *, PT: T#1MS) --- (R Axis8_Halt) (S M3) (R M20)
NETWORK 5
	[M3] - [/Total_Pause] --- (S M4) (S Axis8_Home)
NETWORK 6
	[M4] - [Axis8_Negative_Limit] - DOWN1:F_TRIG(CLK: *) --- (R Axis8_Negative_Invalid)
NETWORK 7
	[M4] - [Axis8_Home_Function.Done] --- (S Axis8_BackHome_OK) (R Axis8_Home) (R Axis8_BackHome_trigger) (R M4) (R M3)
NETWORK 8
	[Total_Pause] - [Axis8_BackHome_trigger] --- (R Axis8_Home) (R Axis8_PTF) (R M4) (R M3) (R M2) (S Axis8_Negative_Invalid) (R Axis8_BackHome_OK) (S M1) (R M20)
NETWORK 9
	*
NETWORK 10
	[Total_Emergency] --- (R M1) (R M20) (R M2) (R M3) (R M4) (R Axis8_BackHome_trigger) (R Axis8_Negative_Invalid) (R Axis8_PTF) (R Axis8_BackHome_OK) (R Axis8_Home)
_END_LD_
(* the same logic as Structured Text *)
(* Network 1 *)
UP1(CLK := Axis8_BackHome_trigger);
IF UP1.Q THEN M1 := TRUE; Axis8_Negative_Invalid := TRUE; END_IF;
(* Network 2 *)
_p1 := M1 AND NOT Total_Pause;
IF _p1 THEN Axis8_PTF := TRUE; M2 := TRUE; M1 := FALSE; END_IF;
(* Network 3 *)
_p2 := M2 AND Axis8_Negative_Limit;
IF _p2 THEN Axis8_Halt := TRUE; M2 := FALSE; M20 := TRUE; Axis8_PTF := FALSE; END_IF;
(* Network 4 *)
T1(IN := M20 AND Axis8_Halt_Function.Done, PT := T#1MS);
IF T1.Q THEN Axis8_Halt := FALSE; M3 := TRUE; M20 := FALSE; END_IF;
(* Network 5 *)
IF M3 AND NOT Total_Pause THEN M4 := TRUE; Axis8_Home := TRUE; END_IF;
(* Network 6 *)
DOWN1(CLK := M4 AND Axis8_Negative_Limit);
IF DOWN1.Q THEN Axis8_Negative_Invalid := FALSE; END_IF;
(* Network 7 *)
_p3 := M4 AND Axis8_Home_Function.Done;
IF _p3 THEN Axis8_BackHome_OK := TRUE; Axis8_Home := FALSE; Axis8_BackHome_trigger := FALSE; M4 := FALSE; M3 := FALSE; END_IF;
(* Network 8 *)
IF Total_Pause AND Axis8_BackHome_trigger THEN Axis8_Home := FALSE; Axis8_PTF := FALSE; M4 := FALSE; M3 := FALSE; M2 := FALSE; Axis8_Negative_Invalid := TRUE; Axis8_BackHome_OK := FALSE; M1 := TRUE; M20 := FALSE; END_IF;
(* Network 9 *)
(* Network 10 *)
IF Total_Emergency THEN M1 := FALSE; M20 := FALSE; M2 := FALSE; M3 := FALSE; M4 := FALSE; Axis8_BackHome_trigger := FALSE; Axis8_Negative_Invalid := FALSE; Axis8_PTF := FALSE; Axis8_BackHome_OK := FALSE; Axis8_Home := FALSE; END_IF;
END_PROGRAM

(* POU Other_Folder/Home_Back/Axis9_Home_Back, LD *)
PROGRAM Axis9_Home_Back
VAR
	UP1: R_TRIG;
	M1: BOOL;
	M2: BOOL;
	UP2: R_TRIG;
	T1: TON;
	M3: BOOL;
	M4: BOOL;
	DOWN1: F_TRIG;
	M20: BOOL;
END_VAR
VAR (* helpers for the ST form of the networks *)
	_p1 : BOOL;
	_p2 : BOOL;
	_p3 : BOOL;
END_VAR
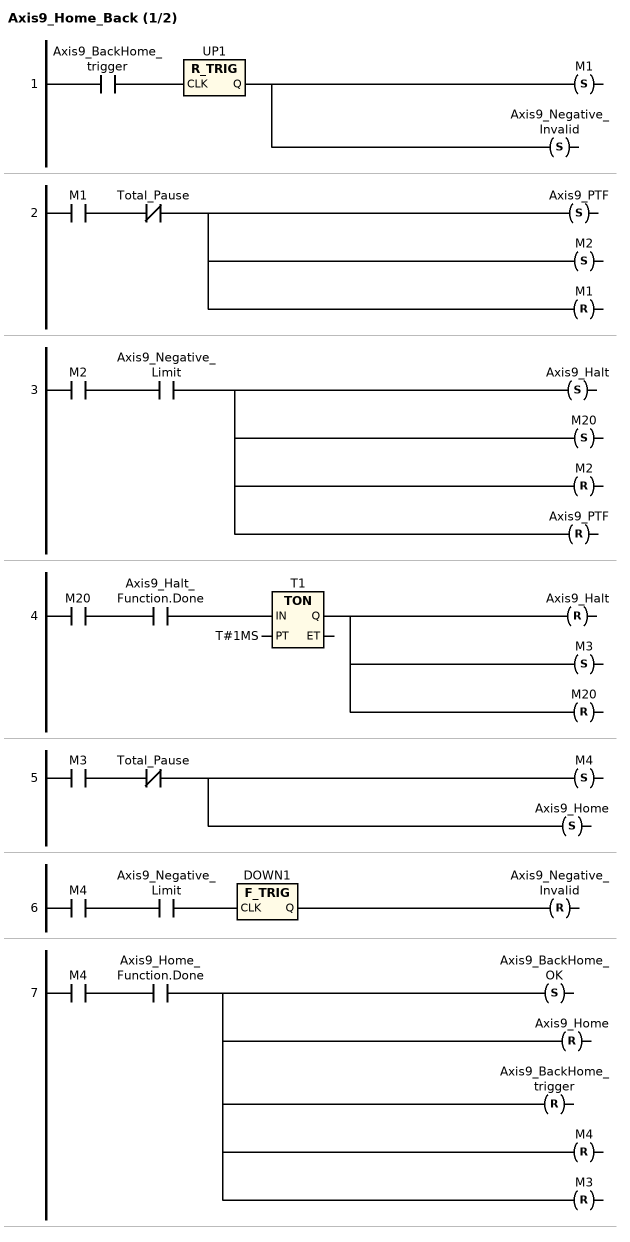
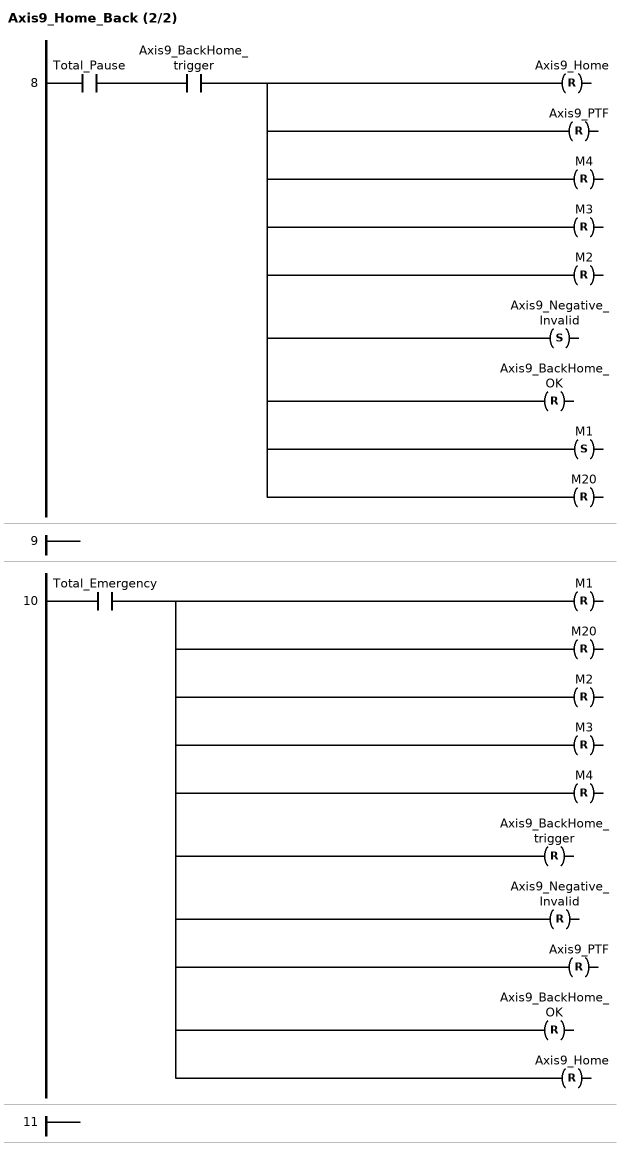
_LD_ (* Ladder Diagram *)
NETWORK 1
	[Axis9_BackHome_trigger] - UP1:R_TRIG(CLK: *) --- (S M1) (S Axis9_Negative_Invalid)
NETWORK 2
	[M1] - [/Total_Pause] --- (S Axis9_PTF) (S M2) (R M1)
NETWORK 3
	[M2] - [Axis9_Negative_Limit] --- (S Axis9_Halt) (S M20) (R M2) (R Axis9_PTF)
NETWORK 4
	[M20] - [Axis9_Halt_Function.Done] - T1:TON(IN: *, PT: T#1MS) --- (R Axis9_Halt) (S M3) (R M20)
NETWORK 5
	[M3] - [/Total_Pause] --- (S M4) (S Axis9_Home)
NETWORK 6
	[M4] - [Axis9_Negative_Limit] - DOWN1:F_TRIG(CLK: *) --- (R Axis9_Negative_Invalid)
NETWORK 7
	[M4] - [Axis9_Home_Function.Done] --- (S Axis9_BackHome_OK) (R Axis9_Home) (R Axis9_BackHome_trigger) (R M4) (R M3)
NETWORK 8
	[Total_Pause] - [Axis9_BackHome_trigger] --- (R Axis9_Home) (R Axis9_PTF) (R M4) (R M3) (R M2) (S Axis9_Negative_Invalid) (R Axis9_BackHome_OK) (S M1) (R M20)
NETWORK 9
	*
NETWORK 10
	[Total_Emergency] --- (R M1) (R M20) (R M2) (R M3) (R M4) (R Axis9_BackHome_trigger) (R Axis9_Negative_Invalid) (R Axis9_PTF) (R Axis9_BackHome_OK) (R Axis9_Home)
NETWORK 11
	*
_END_LD_
(* the same logic as Structured Text *)
(* Network 1 *)
UP1(CLK := Axis9_BackHome_trigger);
IF UP1.Q THEN M1 := TRUE; Axis9_Negative_Invalid := TRUE; END_IF;
(* Network 2 *)
_p1 := M1 AND NOT Total_Pause;
IF _p1 THEN Axis9_PTF := TRUE; M2 := TRUE; M1 := FALSE; END_IF;
(* Network 3 *)
_p2 := M2 AND Axis9_Negative_Limit;
IF _p2 THEN Axis9_Halt := TRUE; M20 := TRUE; M2 := FALSE; Axis9_PTF := FALSE; END_IF;
(* Network 4 *)
T1(IN := M20 AND Axis9_Halt_Function.Done, PT := T#1MS);
IF T1.Q THEN Axis9_Halt := FALSE; M3 := TRUE; M20 := FALSE; END_IF;
(* Network 5 *)
IF M3 AND NOT Total_Pause THEN M4 := TRUE; Axis9_Home := TRUE; END_IF;
(* Network 6 *)
DOWN1(CLK := M4 AND Axis9_Negative_Limit);
IF DOWN1.Q THEN Axis9_Negative_Invalid := FALSE; END_IF;
(* Network 7 *)
_p3 := M4 AND Axis9_Home_Function.Done;
IF _p3 THEN Axis9_BackHome_OK := TRUE; Axis9_Home := FALSE; Axis9_BackHome_trigger := FALSE; M4 := FALSE; M3 := FALSE; END_IF;
(* Network 8 *)
IF Total_Pause AND Axis9_BackHome_trigger THEN Axis9_Home := FALSE; Axis9_PTF := FALSE; M4 := FALSE; M3 := FALSE; M2 := FALSE; Axis9_Negative_Invalid := TRUE; Axis9_BackHome_OK := FALSE; M1 := TRUE; M20 := FALSE; END_IF;
(* Network 9 *)
(* Network 10 *)
IF Total_Emergency THEN M1 := FALSE; M20 := FALSE; M2 := FALSE; M3 := FALSE; M4 := FALSE; Axis9_BackHome_trigger := FALSE; Axis9_Negative_Invalid := FALSE; Axis9_PTF := FALSE; Axis9_BackHome_OK := FALSE; Axis9_Home := FALSE; END_IF;
(* Network 11 *)
END_PROGRAM

(* POU Other_Folder/Home_Back/Axis10_Home_Back, LD *)
PROGRAM Axis10_Home_Back
VAR
	UP1: R_TRIG;
	M1: BOOL;
	M2: BOOL;
	UP2: R_TRIG;
	T1: TON;
	M3: BOOL;
	M4: BOOL;
	DOWN1: F_TRIG;
	M20: BOOL;
END_VAR
VAR (* helpers for the ST form of the networks *)
	_p1 : BOOL;
	_p2 : BOOL;
	_p3 : BOOL;
END_VAR
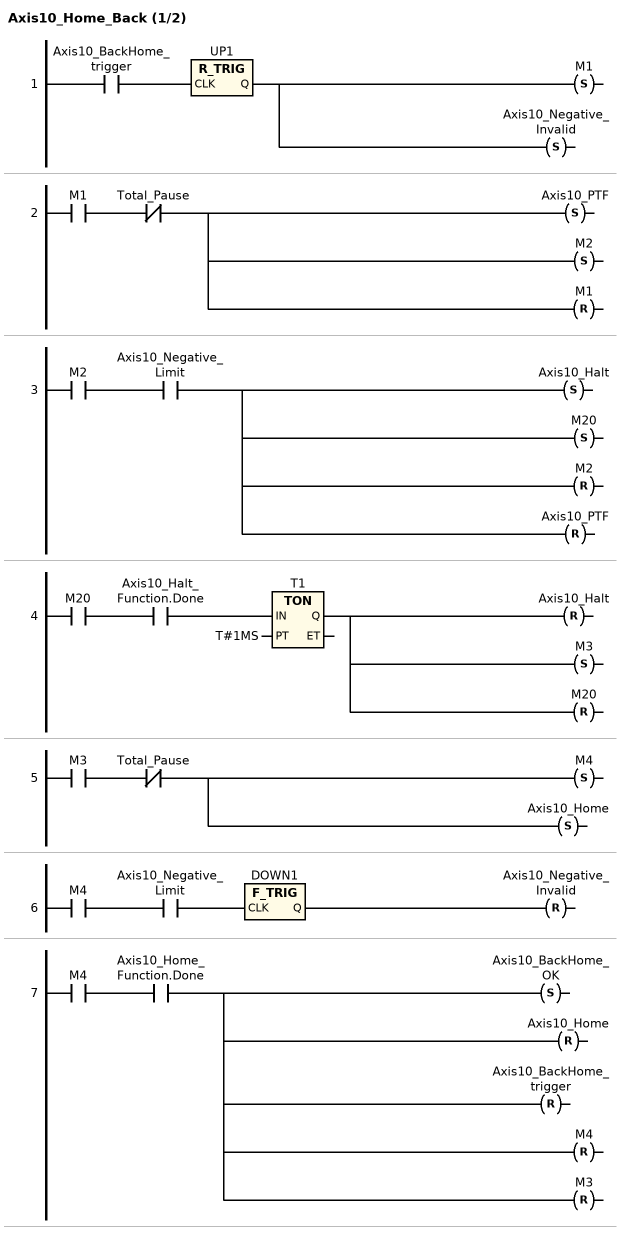
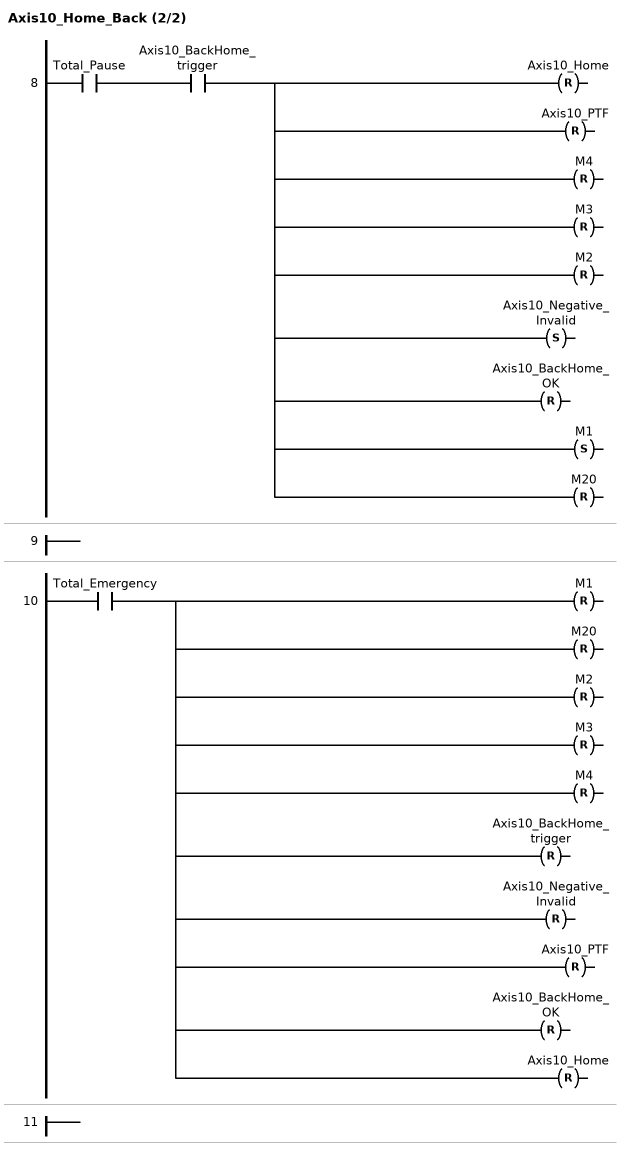
_LD_ (* Ladder Diagram *)
NETWORK 1
	[Axis10_BackHome_trigger] - UP1:R_TRIG(CLK: *) --- (S M1) (S Axis10_Negative_Invalid)
NETWORK 2
	[M1] - [/Total_Pause] --- (S Axis10_PTF) (S M2) (R M1)
NETWORK 3
	[M2] - [Axis10_Negative_Limit] --- (S Axis10_Halt) (S M20) (R M2) (R Axis10_PTF)
NETWORK 4
	[M20] - [Axis10_Halt_Function.Done] - T1:TON(IN: *, PT: T#1MS) --- (R Axis10_Halt) (S M3) (R M20)
NETWORK 5
	[M3] - [/Total_Pause] --- (S M4) (S Axis10_Home)
NETWORK 6
	[M4] - [Axis10_Negative_Limit] - DOWN1:F_TRIG(CLK: *) --- (R Axis10_Negative_Invalid)
NETWORK 7
	[M4] - [Axis10_Home_Function.Done] --- (S Axis10_BackHome_OK) (R Axis10_Home) (R Axis10_BackHome_trigger) (R M4) (R M3)
NETWORK 8
	[Total_Pause] - [Axis10_BackHome_trigger] --- (R Axis10_Home) (R Axis10_PTF) (R M4) (R M3) (R M2) (S Axis10_Negative_Invalid) (R Axis10_BackHome_OK) (S M1) (R M20)
NETWORK 9
	*
NETWORK 10
	[Total_Emergency] --- (R M1) (R M20) (R M2) (R M3) (R M4) (R Axis10_BackHome_trigger) (R Axis10_Negative_Invalid) (R Axis10_PTF) (R Axis10_BackHome_OK) (R Axis10_Home)
NETWORK 11
	*
_END_LD_
(* the same logic as Structured Text *)
(* Network 1 *)
UP1(CLK := Axis10_BackHome_trigger);
IF UP1.Q THEN M1 := TRUE; Axis10_Negative_Invalid := TRUE; END_IF;
(* Network 2 *)
_p1 := M1 AND NOT Total_Pause;
IF _p1 THEN Axis10_PTF := TRUE; M2 := TRUE; M1 := FALSE; END_IF;
(* Network 3 *)
_p2 := M2 AND Axis10_Negative_Limit;
IF _p2 THEN Axis10_Halt := TRUE; M20 := TRUE; M2 := FALSE; Axis10_PTF := FALSE; END_IF;
(* Network 4 *)
T1(IN := M20 AND Axis10_Halt_Function.Done, PT := T#1MS);
IF T1.Q THEN Axis10_Halt := FALSE; M3 := TRUE; M20 := FALSE; END_IF;
(* Network 5 *)
IF M3 AND NOT Total_Pause THEN M4 := TRUE; Axis10_Home := TRUE; END_IF;
(* Network 6 *)
DOWN1(CLK := M4 AND Axis10_Negative_Limit);
IF DOWN1.Q THEN Axis10_Negative_Invalid := FALSE; END_IF;
(* Network 7 *)
_p3 := M4 AND Axis10_Home_Function.Done;
IF _p3 THEN Axis10_BackHome_OK := TRUE; Axis10_Home := FALSE; Axis10_BackHome_trigger := FALSE; M4 := FALSE; M3 := FALSE; END_IF;
(* Network 8 *)
IF Total_Pause AND Axis10_BackHome_trigger THEN Axis10_Home := FALSE; Axis10_PTF := FALSE; M4 := FALSE; M3 := FALSE; M2 := FALSE; Axis10_Negative_Invalid := TRUE; Axis10_BackHome_OK := FALSE; M1 := TRUE; M20 := FALSE; END_IF;
(* Network 9 *)
(* Network 10 *)
IF Total_Emergency THEN M1 := FALSE; M20 := FALSE; M2 := FALSE; M3 := FALSE; M4 := FALSE; Axis10_BackHome_trigger := FALSE; Axis10_Negative_Invalid := FALSE; Axis10_PTF := FALSE; Axis10_BackHome_OK := FALSE; Axis10_Home := FALSE; END_IF;
(* Network 11 *)
END_PROGRAM

(* POU Other_Folder/Home_Back/Axis11_Home_Back, LD *)
PROGRAM Axis11_Home_Back
VAR
	UP1: R_TRIG;
	M1: BOOL;
	M2: BOOL;
	UP2: R_TRIG;
	T1: TON;
	M3: BOOL;
	M4: BOOL;
	DOWN1: F_TRIG;
	M20: BOOL;
END_VAR
VAR (* helpers for the ST form of the networks *)
	_p1 : BOOL;
	_p2 : BOOL;
	_p3 : BOOL;
END_VAR
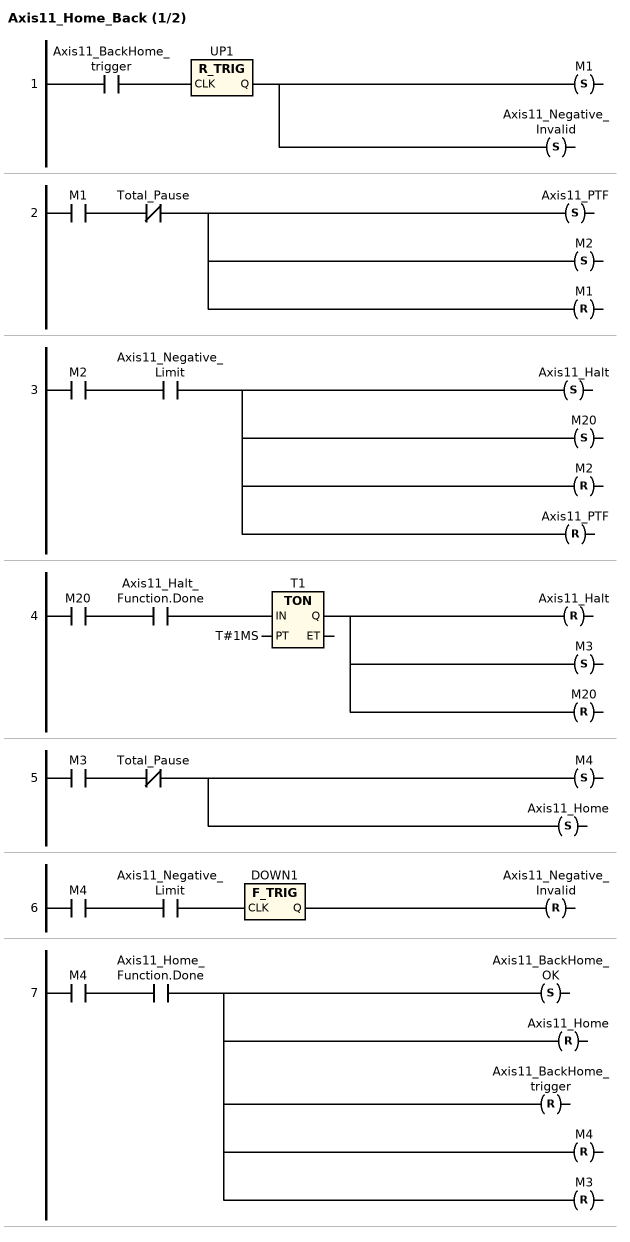
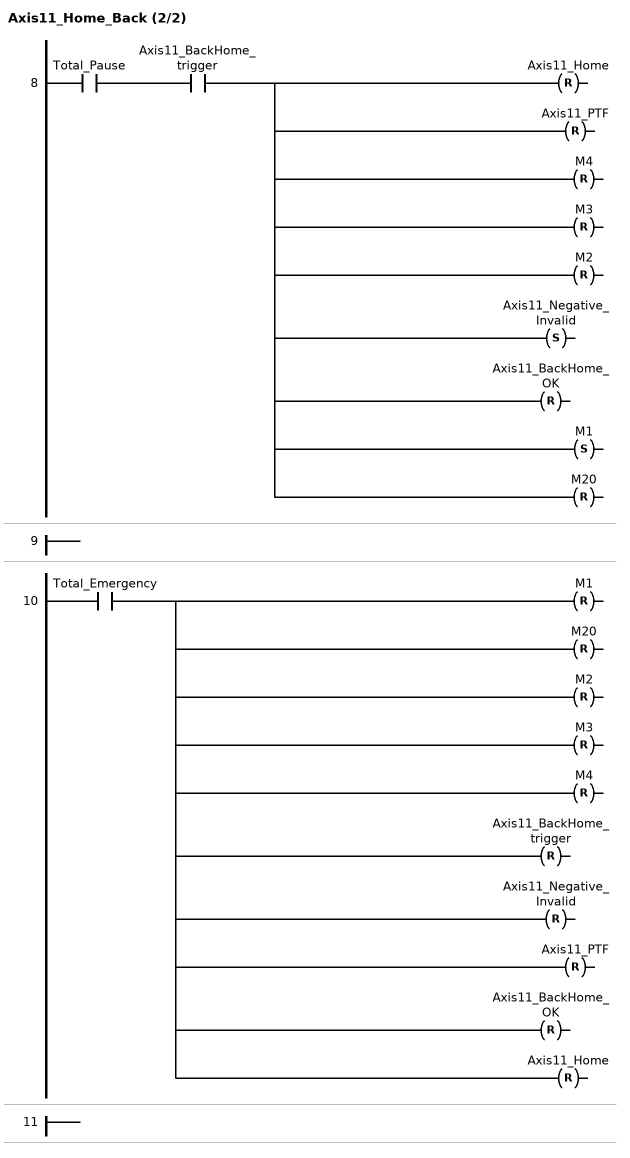
_LD_ (* Ladder Diagram *)
NETWORK 1
	[Axis11_BackHome_trigger] - UP1:R_TRIG(CLK: *) --- (S M1) (S Axis11_Negative_Invalid)
NETWORK 2
	[M1] - [/Total_Pause] --- (S Axis11_PTF) (S M2) (R M1)
NETWORK 3
	[M2] - [Axis11_Negative_Limit] --- (S Axis11_Halt) (S M20) (R M2) (R Axis11_PTF)
NETWORK 4
	[M20] - [Axis11_Halt_Function.Done] - T1:TON(IN: *, PT: T#1MS) --- (R Axis11_Halt) (S M3) (R M20)
NETWORK 5
	[M3] - [/Total_Pause] --- (S M4) (S Axis11_Home)
NETWORK 6
	[M4] - [Axis11_Negative_Limit] - DOWN1:F_TRIG(CLK: *) --- (R Axis11_Negative_Invalid)
NETWORK 7
	[M4] - [Axis11_Home_Function.Done] --- (S Axis11_BackHome_OK) (R Axis11_Home) (R Axis11_BackHome_trigger) (R M4) (R M3)
NETWORK 8
	[Total_Pause] - [Axis11_BackHome_trigger] --- (R Axis11_Home) (R Axis11_PTF) (R M4) (R M3) (R M2) (S Axis11_Negative_Invalid) (R Axis11_BackHome_OK) (S M1) (R M20)
NETWORK 9
	*
NETWORK 10
	[Total_Emergency] --- (R M1) (R M20) (R M2) (R M3) (R M4) (R Axis11_BackHome_trigger) (R Axis11_Negative_Invalid) (R Axis11_PTF) (R Axis11_BackHome_OK) (R Axis11_Home)
NETWORK 11
	*
_END_LD_
(* the same logic as Structured Text *)
(* Network 1 *)
UP1(CLK := Axis11_BackHome_trigger);
IF UP1.Q THEN M1 := TRUE; Axis11_Negative_Invalid := TRUE; END_IF;
(* Network 2 *)
_p1 := M1 AND NOT Total_Pause;
IF _p1 THEN Axis11_PTF := TRUE; M2 := TRUE; M1 := FALSE; END_IF;
(* Network 3 *)
_p2 := M2 AND Axis11_Negative_Limit;
IF _p2 THEN Axis11_Halt := TRUE; M20 := TRUE; M2 := FALSE; Axis11_PTF := FALSE; END_IF;
(* Network 4 *)
T1(IN := M20 AND Axis11_Halt_Function.Done, PT := T#1MS);
IF T1.Q THEN Axis11_Halt := FALSE; M3 := TRUE; M20 := FALSE; END_IF;
(* Network 5 *)
IF M3 AND NOT Total_Pause THEN M4 := TRUE; Axis11_Home := TRUE; END_IF;
(* Network 6 *)
DOWN1(CLK := M4 AND Axis11_Negative_Limit);
IF DOWN1.Q THEN Axis11_Negative_Invalid := FALSE; END_IF;
(* Network 7 *)
_p3 := M4 AND Axis11_Home_Function.Done;
IF _p3 THEN Axis11_BackHome_OK := TRUE; Axis11_Home := FALSE; Axis11_BackHome_trigger := FALSE; M4 := FALSE; M3 := FALSE; END_IF;
(* Network 8 *)
IF Total_Pause AND Axis11_BackHome_trigger THEN Axis11_Home := FALSE; Axis11_PTF := FALSE; M4 := FALSE; M3 := FALSE; M2 := FALSE; Axis11_Negative_Invalid := TRUE; Axis11_BackHome_OK := FALSE; M1 := TRUE; M20 := FALSE; END_IF;
(* Network 9 *)
(* Network 10 *)
IF Total_Emergency THEN M1 := FALSE; M20 := FALSE; M2 := FALSE; M3 := FALSE; M4 := FALSE; Axis11_BackHome_trigger := FALSE; Axis11_Negative_Invalid := FALSE; Axis11_PTF := FALSE; Axis11_BackHome_OK := FALSE; Axis11_Home := FALSE; END_IF;
(* Network 11 *)
END_PROGRAM

(* POU Other_Folder/Home_Back/Axis21_Home_Back, LD *)
PROGRAM Axis21_Home_Back
VAR
	UP1: R_TRIG;
	M1: BOOL;
	M2: BOOL;
	UP2: R_TRIG;
	T1: TON;
	M3: BOOL;
	M4: BOOL;
	DOWN1: F_TRIG;
	M20: BOOL;
END_VAR
VAR (* helpers for the ST form of the networks *)
	_p1 : BOOL;
	_p2 : BOOL;
	_p3 : BOOL;
END_VAR
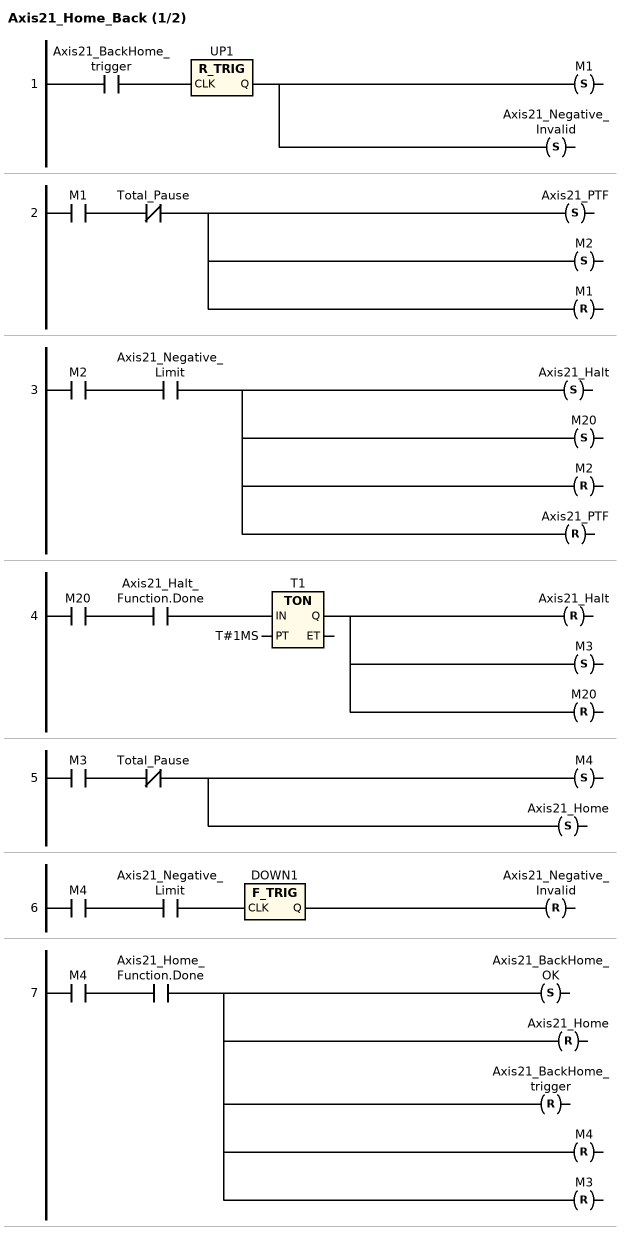
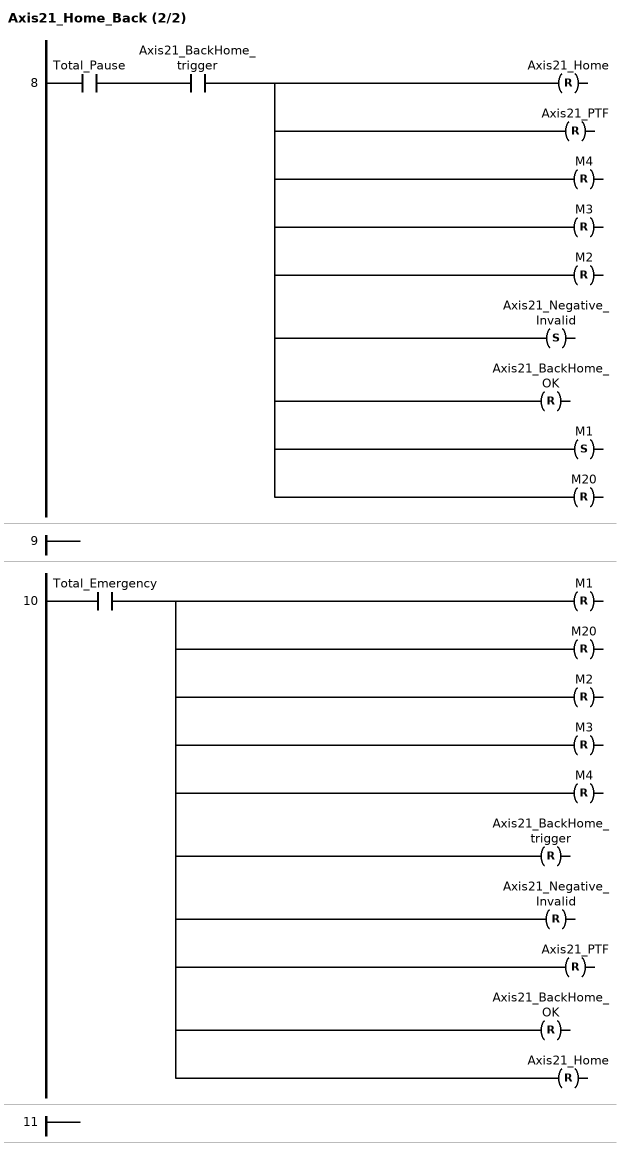
_LD_ (* Ladder Diagram *)
NETWORK 1
	[Axis21_BackHome_trigger] - UP1:R_TRIG(CLK: *) --- (S M1) (S Axis21_Negative_Invalid)
NETWORK 2
	[M1] - [/Total_Pause] --- (S Axis21_PTF) (S M2) (R M1)
NETWORK 3
	[M2] - [Axis21_Negative_Limit] --- (S Axis21_Halt) (S M20) (R M2) (R Axis21_PTF)
NETWORK 4
	[M20] - [Axis21_Halt_Function.Done] - T1:TON(IN: *, PT: T#1MS) --- (R Axis21_Halt) (S M3) (R M20)
NETWORK 5
	[M3] - [/Total_Pause] --- (S M4) (S Axis21_Home)
NETWORK 6
	[M4] - [Axis21_Negative_Limit] - DOWN1:F_TRIG(CLK: *) --- (R Axis21_Negative_Invalid)
NETWORK 7
	[M4] - [Axis21_Home_Function.Done] --- (S Axis21_BackHome_OK) (R Axis21_Home) (R Axis21_BackHome_trigger) (R M4) (R M3)
NETWORK 8
	[Total_Pause] - [Axis21_BackHome_trigger] --- (R Axis21_Home) (R Axis21_PTF) (R M4) (R M3) (R M2) (S Axis21_Negative_Invalid) (R Axis21_BackHome_OK) (S M1) (R M20)
NETWORK 9
	*
NETWORK 10
	[Total_Emergency] --- (R M1) (R M20) (R M2) (R M3) (R M4) (R Axis21_BackHome_trigger) (R Axis21_Negative_Invalid) (R Axis21_PTF) (R Axis21_BackHome_OK) (R Axis21_Home)
NETWORK 11
	*
_END_LD_
(* the same logic as Structured Text *)
(* Network 1 *)
UP1(CLK := Axis21_BackHome_trigger);
IF UP1.Q THEN M1 := TRUE; Axis21_Negative_Invalid := TRUE; END_IF;
(* Network 2 *)
_p1 := M1 AND NOT Total_Pause;
IF _p1 THEN Axis21_PTF := TRUE; M2 := TRUE; M1 := FALSE; END_IF;
(* Network 3 *)
_p2 := M2 AND Axis21_Negative_Limit;
IF _p2 THEN Axis21_Halt := TRUE; M20 := TRUE; M2 := FALSE; Axis21_PTF := FALSE; END_IF;
(* Network 4 *)
T1(IN := M20 AND Axis21_Halt_Function.Done, PT := T#1MS);
IF T1.Q THEN Axis21_Halt := FALSE; M3 := TRUE; M20 := FALSE; END_IF;
(* Network 5 *)
IF M3 AND NOT Total_Pause THEN M4 := TRUE; Axis21_Home := TRUE; END_IF;
(* Network 6 *)
DOWN1(CLK := M4 AND Axis21_Negative_Limit);
IF DOWN1.Q THEN Axis21_Negative_Invalid := FALSE; END_IF;
(* Network 7 *)
_p3 := M4 AND Axis21_Home_Function.Done;
IF _p3 THEN Axis21_BackHome_OK := TRUE; Axis21_Home := FALSE; Axis21_BackHome_trigger := FALSE; M4 := FALSE; M3 := FALSE; END_IF;
(* Network 8 *)
IF Total_Pause AND Axis21_BackHome_trigger THEN Axis21_Home := FALSE; Axis21_PTF := FALSE; M4 := FALSE; M3 := FALSE; M2 := FALSE; Axis21_Negative_Invalid := TRUE; Axis21_BackHome_OK := FALSE; M1 := TRUE; M20 := FALSE; END_IF;
(* Network 9 *)
(* Network 10 *)
IF Total_Emergency THEN M1 := FALSE; M20 := FALSE; M2 := FALSE; M3 := FALSE; M4 := FALSE; Axis21_BackHome_trigger := FALSE; Axis21_Negative_Invalid := FALSE; Axis21_PTF := FALSE; Axis21_BackHome_OK := FALSE; Axis21_Home := FALSE; END_IF;
(* Network 11 *)
END_PROGRAM

(* POU Other_Folder/Home_Back/Axis22_Home_Back, LD *)
PROGRAM Axis22_Home_Back
VAR
	UP1: R_TRIG;
	M1: BOOL;
	M2: BOOL;
	UP2: R_TRIG;
	T1: TON;
	M3: BOOL;
	M4: BOOL;
	DOWN1: F_TRIG;
	M20: BOOL;
END_VAR
VAR (* helpers for the ST form of the networks *)
	_p1 : BOOL;
	_p2 : BOOL;
	_p3 : BOOL;
END_VAR
